(* CoDeSys 2.3 library: Mio_plc.lib *)

(* Global variable list: Globale_Variablen *)
(*
 PLC1131-Library with Functions to M-IO-Handler and IO-Hardware
 Copyright: G.Bachmann GmbH, 1997-2017, Feldkirch - Austria
*)
VAR_GLOBAL CONSTANT
	MIO_PLC_LIBVER					:	STRING(16) 	:=	'V1.39 Release';	(* Version String *)
    MIO_PLC_MMPREADY                :   BOOL        :=  TRUE;               (* MMP Ready *)

	(* Error-Return-Codes *)
	(* ATTENTION: actual Codes must be interpreted (modulo 1000)! *)
	Mio_ERC_Other:			DINT := -1;			(* MIO-Function unsuccessfull *)
	Mio_ERC_ParmInvalid:	DINT := -2;			(* Parameters are invalid *)
	Mio_ERC_NoCard:			DINT := -3;			(* Card not found / existing *)
	Mio_ERC_NoSelf:			DINT := -8;			(* Caller is no PLC *)
	Mio_ERC_Other2:			DINT := -9;			(* MIO-Function unsuccessfull *)
    Mio_ERC_NoMemory:       DINT := -10;		(* Memory can't be allocated *)
	Mio_ERC_Internal:		DINT := -11;		(* Internal Error *)

	(* Constants used with Mio...Select *)
	Mio_OBJ_AllChan:		DWORD := 16#80000000;
	Mio_OBJ_Card:			DWORD := 16#80000001;

    (* possible values for Card-Mode *)
    MIO_MODE_REAL:          DINT := 1;          (* IO-Module is present *)
    MIO_MODE_VIRTUAL:       DINT := 2;          (* IO-Module is virtuel *)
    MIO_MODE_VIRTSIM:       DINT := 3;          (* @deprecated IO-Module has simulated values *)
    MIO_MODE_REALFB:        DINT := 4;          (* IO-Module AT fieldbus *)
    MIO_MODE_VIRTUALRW:     DINT := 5;          (* virtual IO-Module, writeable inputs *)
    MIO_MODE_REALSRV:       DINT := 6;          (* IO-Module connected TO a service *)
    MIO_MODE_VIRTUALSRV:    DINT := 7;          (* IO-Module connected TO a service *)

	(* Constants used as Card-Type *)
	Mio_TYP_MP213:			DINT := 1; 		(* Module of type MP213 *)
	Mio_TYP_MP2XX:			DINT := 1; 		(* Module of type MP2XX *)
	Mio_TYP_DI216:			DINT := 2; 		(* Module of type DI216 *)
	Mio_TYP_DO216:			DINT := 3; 		(* Module of type DO216 *)
	Mio_TYP_DI232:			DINT := 4; 		(* Module of type DI232 *)
	Mio_TYP_DO232:			DINT := 5; 		(* Module of type DO232 *)
	Mio_TYP_AI204:			DINT := 6; 		(* Module of type AI204 *)
	Mio_TYP_AO202:			DINT := 7; 		(* Module of type AO202 *)
	Mio_TYP_ISI202:			DINT := 8; 		(* Module of type ISI202 *)
	Mio_TYP_AIO288:			DINT := 9; 		(* Module of type AIO288 *)
	Mio_TYP_FBM201:			DINT := 10; 	(* Module of type FM201 *)
	Mio_TYP_FBS202:			DINT := 11;		(* Module of type FS202 *)
	Mio_TYP_CM202:			DINT := 12;		(* Module of type CM202 *)
	Mio_TYP_BEM201:			DINT := 13;		(* Module of type BEM201 *)
	Mio_TYP_BES202:			DINT := 14;		(* Module of type BES202 *)
	Mio_TYP_ACR222:			DINT := 15;		(* Module of type ACR222 *)
	Mio_TYP_ME203:			DINT := 16;		(* Module of type ME203 *)
	Mio_TYP_CS200:			DINT := 17;		(* Module of type CS200 *)
	Mio_TYP_RS204:			DINT := 18;		(* Module of type RS204 *)
	Mio_TYP_DMS202:			DINT := 19;		(* Module of type DMS202 *)
	Mio_TYP_NT230:			DINT := 20;		(* Module of type NT230 *)
	Mio_TYP_DIO216:			DINT := 21;		(* Module of type DIO216 *)
	Mio_TYP_DI212:			DINT := 24;		(* Module of type DI212 *)
	Mio_TYP_DIO264_C:		DINT := 25;		(* Module of type DIO16/32/48/64_C *)
	Mio_TYP_BS2XX:			DINT := 26;		(* Bus Module of type BS2XX *)
	Mio_TYP_FM21X:			DINT := 27;		(* Module of type FM211, FM212 *)
	Mio_TYP_FS21X:			DINT := 28;		(* Module of type FS211, FS212 *)
	Mio_Typ_FM2XX:   		DINT := 27; 	(* Module of type FM211, FM212, FM221, FM222 *)
	Mio_Typ_FS2XX:   		DINT := 28;  	(* Module of type FS211, FS212, FS221, FS222 *)
	Mio_TYP_ES200:			DINT := 29;		(* Module of type ES200 *)
	Mio_TYP_DPM200:			DINT := 30;		(* Module of type DPM200 *)
	Mio_TYP_CNT204:			DINT := 31;		(* Module of type CNT204 *)
	Mio_TYP_PTAI216:		DINT := 32;		(* Module of type PTAI216 *)
	Mio_TYP_PWM202:			DINT := 33;		(* Module of type PWM202 *)
	Mio_TYP_TCO216_C:		DINT := 34;		(* Module of type TCO216-C *)
	Mio_TYP_AO208:			DINT := 35;		(* Module of type AO208 *)
	Mio_TYP_DIO280:			DINT := 36;		(* Module of type DIO248/64/80 *)
	Mio_TYP_DIO2XX:			DINT := 36;		(* Module of type DIO248/64/80 *)
	Mio_TYP_TTL264:			DINT := 37;		(* Module of type TTL264 *)
	Mio_TYP_SEM201:         DINT := 38;     (* Module of type SEM201 *)
	Mio_TYP_IOP201:         DINT := 39;     (* Module of type IOP201 *)
    Mio_TYP_BSI200:         DINT := 40;     (* Module of type BSI200 (no drv) *)
    Mio_TYP_MTS200:         DINT := 41;     (* Module of type MTS200 (no drv) *)
    Mio_TYP_PCFS212:        DINT := 42;     (* Module of type PCFS212 *)
    Mio_TYP_DNM201:         DINT := 43;     (* Module of type DNM201 *)
	Mio_TYP_AI20XSI:		DINT := 44;		(* Module of type AI20X/SI *)
	Mio_TYP_AO20XSI:		DINT := 45;		(* Module of type AO20X/SI *)
    Mio_TYP_WT305E:         DINT := 46;     (* Module of type WT305e (no drv) *)
	Mio_TYP_EM203:			DINT := 47; 	(* Module of type EM203 *)
	Mio_TYP_MPC2XX:			DINT := 49; 	(* Module of type MPC2XX *)
	Mio_TYP_MX2XX:			DINT := 50;		(* Module of type MX2XX *)
	Mio_TYP_WT3XX:          DINT := 51;     (* Module of type WT3XX (no drv) *)
    Mio_TYP_PCM201:         DINT := 52;     (* Internal Module (no drv) *)
    Mio_TYP_DIO232:         DINT := 53;     (* Module of type DIO232 *)
    Mio_TYP_BET200:         DINT := 54;     (* Internal Module (no drv) *)
    Mio_TYP_PN201:          DINT := 55;     (* Module of type PN201 *)
    Mio_TYP_NT255:          DINT := 56;     (* Module of type NT255 *)
    Mio_TYP_MBM201:         DINT := 57;     (* Module of type Modbus Master *)
    Mio_TYP_WT2XX:          DINT := 58;     (* Module of type WT2XX (no drv) *)
    Mio_TYP_CT2XX:          DINT := 59;     (* Module of type CT2XX *)
    Mio_TYP_DA3284C:        DINT := 60;     (* Module of type DA3284C *)
	Mio_TYP_AIC2XX:         DINT := 61;     (* Module of type AIC2XX *)
	Mio_TYP_CAN:            DINT := 62;     (* Logical CAN Module *)
	Mio_TYP_ECAT201:        DINT := 63;     (* Module of type ECAT201 *)
	Mio_TYP_TI214:          DINT := 64;     (* Module of type TI214 *)
	Mio_TYP_EVALBOARD:      DINT := 65;     (* HW Evaluation Board *)
	Mio_TYP_PN23:           DINT := 66;     (* PCI Module of type PN23 ProfiNet IRT *)
    Mio_TYP_OT100:          DINT := 67;     (* OT100 Terminal *)
    Mio_TYP_SLC284:         DINT := 68;     (* Module OF TYPE SLC284 *)
    Mio_TYP_SDI208:         DINT := 69;     (* Module OF TYPE SDI208 *)
    Mio_TYP_SDO204:         DINT := 70;     (* Module OF TYPE SDO204 *)
	Mio_TYP_ETH2X:          DINT := 77;     (* Module of type ETH2X *)
	Mio_TYP_DOR206:         DINT := 78;     (* Module of type DOR206 *)
	Mio_TYP_DMW200:         DINT := 79;     (* Module of Drive-Middleware *)
	Mio_TYP_SERCOS:         DINT := 80;     (* Module of Drive-Middleware *)
	Mio_TYP_AP211:          DINT := 81;     (* Module of type AP21X *)
	Mio_TYP_MH2XX:          DINT := 82;     (* Module of type MH2XX *)
	Mio_TYP_MMSCNLT:        DINT := 83;     (* Module of type MMS-Client *)
	Mio_TYP_SFS240C:        DINT := 84;     (* Module of type SFS240C *)
	Mio_TYP_FCS2XX:         DINT := 85;     (* Module of type FCS2xx *)
	Mio_TYP_CT1300:         DINT := 86;     (* Module of type CT1300 *)
	Mio_TYP_OT1300:         DINT := 87;     (* Module of type OT1300 *)
	Mio_TYP_AI208SI:        DINT := 88;     (* Module of type AI208/SI *)
	Mio_TYP_GMP232:         DINT := 89;     (* Module of type GMP232 *)
    Mio_TYP_BCP200:         DINT := 90;     (* Module OF TYPE BCP200 *)
    Mio_TYP_BCH200:         DINT := 91;     (* Module OF TYPE BCH200 *)
    Mio_TYP_EM213:          DINT := 92;     (* Module OF TYPE EM213 *)
    Mio_TYP_ECS200:         DINT := 93;     (* Module OF TYPE ECS200 *)
    Mio_TYP_BCP202:         DINT := 94;     (* Module OF TYPE BCP202 *)
    Mio_TYP_BCH202:         DINT := 95;     (* Module OF TYPE BCH202 *)
    Mio_TYP_BCR202:         DINT := 96;     (* Module OF TYPE BCR202 *)
    Mio_TYP_MC2XX:          DINT := 97;     (* Module OF TYPE MC2XX *)
    Mio_TYP_MBUS:           DINT := 98;     (* Service OF TYPE MBUS *)
	MIO_TYP_GIO2XX:         DINT := 99;     (* Service OF TYPE GIO2XX *)
	MIO_TYP_GSP274:         DINT := 100;    (* Module OF TYPE GSP274 *)
	MIO_TYP_S60870_5:       DINT := 101;    (* Module OF TYPE IEC 60870-5-104 server *)
    MIO_TYP_AIO2XX:         DINT := 102;    (* Module of type AIO2XX *)
	MIO_TYP_SVMXXX:     	DINT := 103;    (* Module of type SVMXXX *)
	MIO_TYP_OPCUAS:      	DINT := 104;    (* Module of type OPCUAS *)
	MIO_TYP_BPC600:       	DINT := 105;    (* Module of type BCP600 *)
	MIO_TYP_STMI3XX:      	DINT := 106;    (* Module of type STMI3XX *)
	MIO_TYP_GM260:       	DINT := 107;    (* Module of type GM260 *)
	MIO_TYP_CPC2XX:         DINT := 108;    (* CompactPLC of type CPC2xx *)
	MIO_TYP_CAIO284:        DINT := 109;    (* AIO284 for CPC2XX *)
	MIO_TYP_CISI2XX:     	DINT := 110;    (* ISI2XX for CPC2XX *)
	MIO_TYP_CDIO2XX:        DINT := 111;    (* DIO2XX for CPC2XX *)
	MIO_TYP_GM2XX:      	DINT := 112;    (* Module of type GM2XX (GM210 and GM230) *)
	MIO_TYP_OT1200:       	DINT := 113;    (* Module of type OT1200 *)
	MIO_TYP_MR2XX:        	DINT := 114;  	(* Module of type MR2XX *)
	MIO_TYP_DIOXXC:       	DINT := 115;    (* Module of type DIOxx-C Standalone CAN-Modules *)
	MIO_TYP_AIO2XXSI:     	DINT := 116;    (* Module of type AIO2XX/SI *)
	MIO_TYP_DNP3:         	DINT := 117;   	(* Service of type DNP3 *)
	MIO_TYP_SCT202:         DINT := 118;    (* Module of type SCT202 *)
	MIO_TYP_GMP232X:      	DINT  := 119;   (* Module of type GMP232/X *)
	MIO_TYP_PVA2XX:       	DINT  := 120;   (* Module of type PVA2XX *)
	MIO_TYP_TSTDRV:       	DINT  := 254;   (* Generic ID for test drivers *)

    (* Constants used as Card-Variant *)

	(* in case of type MIO_TYP_MP2XX *)
	MIO_V_MP213:    DINT  := 0;     (* Module of type MP213 *)
	MIO_V_MP226:    DINT  := 1;     (* Module of type MP226 *)
	MIO_V_MP236:    DINT  := 2;     (* Module of type MP236 *)
	MIO_V_MP240:    DINT  := 3;     (* Module of type MP240 *)
	MIO_V_MP213EW:  DWORD := 16#20; (* Module of type MP213/EW *)
	MIO_V_MP226EW:  DWORD := 16#21; (* Module of type MP226/EW *)

	(* in case of type MIO_TYP_ME203 *)
	MIO_V_ME203:    DINT  := 0;     (* Module of type ME203 *)
	MIO_V_ME203N:   DINT  := 1;     (* Module of type ME203/N *)
	MIO_V_ME203C:   DINT  := 2;     (* Module of type ME203/C *)
	MIO_V_ME203CN:  DINT  := 3;     (* Module of type ME203/CN *)
	MIO_V_ME203E:   DINT  := 4;     (* Module of type ME203/E *)
	MIO_V_ME203EN:  DINT  := 5;     (* Module of type ME203/EN *)
	MIO_V_ME203CNW: DWORD := 16#23; (* Module of type ME203/CNW *)

	(* WT/CT Version in case of type Mio_TYP_WTXXX for 200 and 300 series. *)
	MIO_VF_DISPLAYMASK: DWORD := 16#0f;         (* filter for display type *)
	MIO_VF_DIMMABLE:    DWORD := 16#10;         (* dimmable display *)
	MIO_VF_IRTOUCH:     DWORD := 16#40;         (* IR Touch *)
	MIO_VF_ALARM:       DWORD := 16#80;         (* has extern alarm IOs *)
	MIO_V_WT305:        DINT  := 0;             (* Module of type WT305 1/4 VGA *)
	MIO_V_WT306:        DINT  := 1;             (* Module of type WT306 VGA *)
	MIO_V_WT310:        DINT  := 2;             (* Module of type WT310 *)
	MIO_V_WT312:        DINT  := 3;             (* Module of type WT312 *)
	MIO_V_WT315:        DINT  := 4;             (* Module of type WT315 *)
	MIO_V_WT317:        DINT  := 5;             (* Module of type WT317 *)
	MIO_V_WT319:        DINT  := 6;             (* Module of type WT319 *)
	MIO_V_WT305V:       DINT  := 7;             (* Module of type WT305V *)
	MIO_V_CT305:        DINT  := MIO_V_WT305;   (* Module of type CT305 1/4 VGA *)
	MIO_V_CT306:        DINT  := MIO_V_WT306;   (* Module of type CT306 VGA *)
	MIO_V_CT310:        DINT  := MIO_V_WT310;   (* Module of type CT310 *)
	MIO_V_CT312:        DINT  := MIO_V_WT312;   (* Module of type CT312 *)
	MIO_V_CT315:        DINT  := MIO_V_WT315;   (* Module of type CT315 *)
	MIO_V_CT317:        DINT  := MIO_V_WT317;   (* Module of type CT317 *)
	MIO_V_CT319:        DINT  := MIO_V_WT319;   (* Module of type CT319 *)
	MIO_V_CT305V:       DINT  := MIO_V_WT305V;  (* Module of type CT305 VGA *)
	MIO_V_WT205:        DINT  := MIO_V_WT305;   (* Module of type WT205 1/4 VGA *)
	MIO_V_WT205V:       DINT  := MIO_V_WT305V;  (* Module of type WT205 VGA *)
	MIO_V_CT205:        DINT  := MIO_V_WT205;   (* Module of type CT205 1/4 VGA *)
	MIO_V_CT205V:       DINT  := MIO_V_WT205V;  (* Module of type CT205 VGA *)
	MIO_V_CT205M:       DWORD := 16#00000097;

	(* in case of type MIO_TYP_MPC2XX *)
	MIO_V_MPC240:   DINT  := 0;     (* Module of type MPC240 *)
	MIO_V_MPC265:   DINT  := 1;     (* Module of type MPC265 *)
	MIO_V_MPC270:   DINT  := 2;     (* Module of type MPC270 *)
	MIO_V_MPC293:   DINT  := 3;     (* Module of type MPC293 *)
	MIO_V_MPC240CW: DWORD := 16#20; (* Module of type MPC240/CW *)
	MIO_V_MPC265CW: DWORD := 16#21; (* Module of type MPC265/CW *)
	MIO_V_MPC270CW: DWORD := 16#22; (* Module of type MPC270/CW *)
	MIO_V_MPC293CW: DWORD := 16#23; (* Module of type MPC293/CW *)

	(* in case of type MIO_TYP_MPC2XX (MPE2xx CPUs) *)

	MIO_V_MPE2XX:   DWORD := 16#10; (* Module of type MPE2xx *)
	MIO_V_MPE240:   DWORD := 16#10; (* Module of type MPE240 *)
	MIO_V_MPE265:   DWORD := 16#11; (* Module of type MPE265 *)
	MIO_V_MPE270:   DWORD := 16#12; (* Module of type MPE270 *)

	(* in case of type MIO_TYP_MX2XX *)
	MIO_VF_MX2xx_N:     DWORD := 16#01;         (* MX2xx bitmask: has integrated power supply *)
	MIO_VF_MX2xx_CW:    DWORD := 16#20;         (* MX2xx bitmask: is a cold weather variant *)
	MIO_V_MX213:        DWORD := 16#00;         (* MX2xx bitmask: Module of type MX213 *)
	MIO_V_MX213N:       DWORD := 16#00000001;
	MIO_V_MX213CW:      DWORD := 16#00000020;
	MIO_V_MX213NCW:     DWORD := 16#00000021;
	MIO_V_MX207:        DWORD := 16#02;         (* MX2xx bitmask: Module of type MX207 *)
	MIO_V_MX207N:       DWORD := 16#00000003;
	MIO_V_MX207CW:      DWORD := 16#00000022;
	MIO_V_MX207NCW:     DWORD := 16#00000023;
	MIO_V_MX220:        DWORD := 16#04;         (* MX2xx bitmask: Module of type MX220 *)
	MIO_V_MX220N:       DWORD := 16#00000005;
	MIO_V_MX220CW:      DWORD := 16#00000024;
	MIO_V_MX220NCW:     DWORD := 16#00000025;

	(* in case of type MIO_TYP_MH2XX *)
	MIO_V_MH212S:   DINT  := 0; (* Module of type MH212/S *)
	MIO_V_MH212:    DINT  := 1; (* Module of type MH212 *)
	MIO_V_MH230:    DINT  := 2; (* Module of type MH230 *)

	(* in case of type MIO_TYP_MC2XX *)
	MIO_V_MC205:    DINT  := 0; (* Module of type MC205 (600MHz) *)
	MIO_V_MC210:    DINT  := 1; (* Module of type MC210 (1600MHz) *)
	MIO_V_MC206:    DINT  := 2; (* Module OF TYPE MC206 (Single core 800MHz) *)
	MIO_V_MC212:    DINT  := 3; (* Module OF TYPE MC212 (Dual core 1300MHz) *)
	MIO_V_MC220:    DINT  := 4; (* Module OF TYPE MC220 (Quad core 1600MHz) *)

	(* in case of type MIO_TYP_ISI2xx *)
	MIO_V_ISI222:   DWORD := 16#81; (* Module of type ISI222 *)

	(* in case of type MIO_TYP_DIOXXC *)
	MIO_V_DIO43C:   DWORD := 16#00; (* Module of type DIO43-C *)
	MIO_V_DIO62C:   DWORD := 16#01; (* Module of type DIO62-C *)

	(* in case of type MIO_TYP_CPC2XX *)
	MIO_V_CPC210:   DWORD := 16#01; (* Module of type CPC210 *)

	(* in case of type MIO_TYP_MR2XX *)
	MIO_V_MR201:    DWORD := 16#00; (* Module of type MR201 *)
	MIO_V_MR202:    DWORD := 16#01; (* Module of type MR202 *)

	(* in case of type MIO_TYP_GM2XX *)
	MIO_V_GM230:    DWORD := 16#00; (* Module of type GM230 *)
	MIO_V_GM210:    DWORD := 16#01; (* Module of type GM210 *)

	(* in case of type MIO_TYP_GMP232X *)
	MIO_V_GMP232_1: DWORD := 16#01; (* Module of type GMP232/1 *)
	MIO_V_GMP232_2: DWORD := 16#02; (* Module of type GMP232/2 *)
	MIO_V_GMP232_3: DWORD := 16#03; (* Module of type GMP232/3 *)
	MIO_V_GMP232_4: DWORD := 16#04; (* Module of type GMP232/4 *)

    (* Constants used as Card- and Channel-Category *)
	Mio_CTG_Di:				DWORD := 16#0001; 		(* Card/Chan with DI capability *)
	Mio_CTG_Do:				DWORD := 16#0002; 		(* Card/Chan with DO capability *)
	Mio_CTG_Ai:				DWORD := 16#0004; 		(* Card/Chan with AI capability *)
	Mio_CTG_Ao:				DWORD := 16#0008; 		(* Card/Chan with AO capability *)
	Mio_CTG_Inc:			DWORD := 16#0010; 		(* Card/Chan with INC capability *)
	Mio_CTG_Ssi:			DWORD := 16#0020; 		(* Card/Chan with SSI capability *)
	Mio_CTG_Drive:			DWORD := 16#0040; 		(* Card/Chan for drives *)
	Mio_CTG_Interface:		DWORD := 16#0080; 		(* Card/Chan with an interface *)
	Mio_CTG_Count:			DWORD := 16#0100; 		(* Card/Chan with CNT capability *)
	Mio_CTG_Trigg:			DWORD := 16#0200; 		(* Card/Chan with TRG capability *)
	Mio_CTG_Pwm:			DWORD := 16#0400; 		(* Card/Chan with PWM capability *)
	Mio_CTG_Freq:			DWORD := 16#0800; 		(* Card/Chan with FREQ capability *)
	Mio_CTG_Stat:			DWORD := 16#1000; 		(* Card/Chan with Status cap. *)
	Mio_CTG_Cntrl:			DWORD := 16#2000; 		(* Card/Chan with Control cap. *)
	Mio_CTG_Time:			DWORD := 16#8000;		(* Card/Chan with time measure cap. *)
	Mio_CTG_Diff: 			DWORD := 16#10000;		(* Card/Chan with diff. measure cap. *)
    Mio_CTG_Velocity:       DWORD := 16#20000;      (* Card with velocity measure cap. *)
	Mio_CTG_Bes:			DWORD := 16#04000000; 	(* Card is Bus Extension Slave *)
	Mio_CTG_Bem:			DWORD := 16#08000000; 	(* Card is Bus Extension Master *)
	Mio_CTG_Cpu:			DWORD := 16#10000000; 	(* CPU module *)
	Mio_CTG_Fbs:			DWORD := 16#20000000; 	(* Card with FastBusSlave cap. *)
	Mio_CTG_Fbm:			DWORD := 16#40000000; 	(* Card with FastBusMaster cap. *)
	Mio_CTG_FB:				DWORD := 16#80000000; 	(* Card with Fieldbus capability *)

	(* Constants used as Card- and Channel-Flags *)
	Mio_FLG_Read:			DWORD := 16#0001; 		(* Card/Chan is readable *)
	Mio_FLG_Write:			DWORD := 16#0002; 		(* Card/Chan is writable *)
	Mio_FLG_RW:				DWORD := 16#0003; 		(* Card/Chan is read-/writable *)
	Mio_FLG_Error:			DWORD := 16#0004; 		(* Card/Chan has error interrupt *)
	Mio_FLG_Event:			DWORD := 16#0008; 		(* Card/Chan has event interrupt *)
	Mio_FLG_Select:			DWORD := 16#0010; 		(* Card/Chan has select functions *)
	Mio_FLG_BadIO: 			DWORD := 16#0400; 		(* Card has been deactivated *)
	Mio_FLG_Fnled:			DWORD := 16#0800; 		(* Card has function for LED flashing *)
	Mio_FLG_Bcheck:			DWORD := 16#1000; 		(* Card supports IO-Bus check *)
	Mio_FLG_Acheck:			DWORD := 16#2000; 		(* Card supports Alive check *)
	Mio_FLG_Watchdog:		DWORD := 16#4000; 		(* Card has watchdog to be triggered *)
	Mio_FLG_Firmware:		DWORD := 16#8000; 		(* Card has firmware or updatable logic on it *)
	Mio_FLG_SVar:			DWORD := 16#200000;		(* Card has service variables *)
	Mio_FLG_HwPiReady:		DWORD := 16#400000;		(* Card is ready for hardware process image *)
	Mio_FLG_HwPiSupp:		DWORD := 16#800000;		(* Card supports hardware process image *)
	Mio_FLG_FIFOVar:		DWORD := 16#1000000;	(* Card supports variable FIFO flush address *)
	Mio_FLG_ChPiSupp:		DWORD := 16#2000000;	(* Card supports selected channel process image *)

	(* Constants used for Error-State *)
	Mio_ERR_Badstation:		DWORD := 16#0001; 		(* Module is on Bad Station *)
	Mio_ERR_Power:			DWORD := 16#0002;		(* Ext./int. power failure *)
	Mio_ERR_BrokenWire:		DWORD := 16#0004;		(* Open In/Out circuit *)
	Mio_ERR_ShortCirc:		DWORD := 16#0008;		(* Short In/Out circuit *)
	Mio_ERR_TempTooHi:		DWORD := 16#0010;		(* Temperatue too high *)
	Mio_ERR_Decoder:		DWORD := 16#0020;		(* Decoder/Encoder error *)
	Mio_ERR_Accu:			DWORD := 16#0040;		(* @deprecated Battery voltage low *)
    Mio_ERR_ChanDisabled:   DWORD := 16#0040;       (* Channel is disabled *)
	Mio_ERR_Init:			DWORD := 16#0080;		(* @deprecated Error in init function *)
	Mio_ERR_BadConfig:		DWORD := 16#0080;		(* Configuration not valid *)
	Mio_ERR_Watchdog:		DWORD := 16#0100;		(* Internal watchdog error *)
	Mio_ERR_External:		DWORD := 16#0200;		(* External error *)
	Mio_ERR_Ready:			DWORD := 16#0400;		(* @deprecated Modul internal cycle done *)
	Mio_ERR_Dead: 			DWORD := 16#0400; 		(* Module alive test failed *)
	Mio_ERR_OutDisabled:	DWORD := 16#0800;		(* Output is disabled *)
	Mio_ERR_Voltagetohi:	DWORD := 16#1000;		(* External voltage too high *)
	Mio_ERR_Voltagetolo:	DWORD := 16#2000;		(* External voltage too low *)
	Mio_ERR_Currenttohi:	DWORD := 16#4000;		(* Output current too high *)
	Mio_ERR_Badprofile:		DWORD := 16#00008000; 	(* Profile not valid *)
	Mio_ERR_MaskSystem:		DWORD := 16#0000FFFF;	(* Generic errors *)
	Mio_ERR_MaskUser:		DWORD := 16#FFFF0000;	(* Driver specific error *)

	(* Constants used for Event-State *)
	Mio_EVT_Value:			DWORD := 16#0001;		(* Event on change OF value *)
	Mio_EVT_Reference:		DWORD := 16#0002;		(* Event AT reference point *)
	Mio_EVT_Reset:			DWORD := 16#0004;		(* Event home done *)
	Mio_EVT_Latchstrb:		DWORD := 16#0010;		(* Latch into strobe register done *)
	Mio_EVT_Latchref:		DWORD := 16#0020;		(* Latch into reference register done *)
	Mio_EVT_Latchstrbov:	DWORD := 16#0040;		(* Latch strobe overwritten *)
	Mio_EVT_Latchreflos:	DWORD := 16#0080;		(* Latch referenz register lost *)

	(* Constants used as Error-State in case of SSI-Inputs *)
	Mio_ERR_Clock:			DWORD := 16#00010000;

   (* Possible driver specific error for PWM module *)
	MIO_ERR_MAXCURRENT:   DWORD := 16#00040000;   (* Max. current reached *)

   (* Possible driver specific error for PCFS module *)
	MIO_ERR_TRANSMIT: DWORD := 16#00100000;   (* Data transmission error *)
	MIO_ERR_PCIRESET: DWORD := 16#00200000;   (* PCI-Reset *)

   (* Possible driver specific error for AI204/SI module *)
	MIO_ERR_POSRANGE:     DWORD := 16#00400000;   (* Value above maximum *)
	MIO_ERR_NEGRANGE:     DWORD := 16#00800000;   (* Value below minimum *)
	MIO_ERR_MONITORING:   DWORD := 16#01000000;   (* Monitoring error! *)

    (* Possible driver specific error for Safety modules *)
    Mio_ERR_SafetyGenErr:   DWORD := 16#00010000;    (* General module error *)

	(* Possible driver specific errors for MBM201 modules *)
	MIO_ERR_CONNECTION:       DWORD := 16#00000400;   (* No connection *)
	MIO_ERR_EXCEPTION:        DWORD := 16#00010000;   (* Modbus exception *)
	MIO_ERR_CYCLETIMETOOLONG: DWORD := 16#00020000;   (* Cycle time too long *)
	MIO_ERR_CRCERROR:         DWORD := 16#00040000;   (* CRC error *)

   (* Possible driver specific errors/warning for FM2XX/FS2XX, FCS2XX modules *)
	MIO_WRN_LINE_A:     DWORD := 16#00010000;   (* FO Line A RX Power has critical level. *)
	MIO_ERR_LINE_A:     DWORD := 16#00020000;   (* FO Line A RX Power is below critical level. *)
	MIO_WRN_LINE_B:     DWORD := 16#00100000;   (* FO Line B RX Power has critical level. *)
	MIO_ERR_LINE_B:     DWORD := 16#00200000;   (* FO Line B RX Power is below critical level. *)
	MIO_ERR_TRIGGER_A:  DWORD := 16#01000000;   (* FO Line A user defined triggervalue *)

    (* ECS200 specific error and event interrupts *)
    MIO_ERR_ECSGENERR:      DWORD := 16#00010000;     (* General module error *)
    MIO_EVT_ECSSYNC0:       DWORD := 16#00010000;     (* SYNC0 Event *)
    MIO_EVT_ECSSYNC1:       DWORD := 16#00020000;     (* SYNC1 Event *)

    (* DIO2xx specific error and event interrupts *)
    MIO_ERR_PWFMODULE:      DWORD := 16#00020000;     (* Power fail complete module *)
    MIO_ERR_PHASE:          DWORD := 16#00040000;     (* Phase error *)
    MIO_EVT_OVERFLOW:       DWORD := 16#02000000;     (* Value overflow *)

    (* GIO212, AIO216 and AIO208 specific error and event interrupts *)
	MIO_ERR_LOWERRANGE:   DWORD := 16#00010000;       (* Lowerrange exceeded *)
	MIO_ERR_UPPERRANGE:   DWORD := 16#00020000;       (* Upperrange exceeded *)
	MIO_EVT_REFERENCE2:   DWORD := 16#00010000;       (* Second reverence value reached *)
    MIO_EVT_LOWERLIMIT:   DWORD := 16#00020000;       (* Lower LIMIT reached *)
    MIO_EVT_UPPERLIMIT:   DWORD := 16#00040000;       (* Upper LIMIT reached *)

   (* Events for SCT202 module *)
    MIO_EVT_OVERSPEED:    DWORD := 16#00010000;       (* Chan 1-4 *)
    MIO_EVT_STAGNATION:   DWORD := 16#00020000;       (* Chan 1-4 *)

	(* RS204 specific event interrupts *)
	MIO_EVT_POWER_UART1:  DWORD := 16#00010000;   	(* Powerfail UART1 *)
	MIO_EVT_POWER_UART2:  DWORD := 16#00020000;   	(* Powerfail UART2 *)
	MIO_EVT_POWER_UART3:  DWORD := 16#00040000;   	(* Powerfail UART3 *)
	MIO_EVT_POWER_UART4:  DWORD := 16#00080000;   	(* Powerfail UART4 *)

	(* GMP232X specific event flags. None of them are shared with the standard GMP232. *)
	MIO_EVT_QU_PCC1:     DWORD := 16#00000002;   (* QU PCC1 *)
	MIO_EVT_QU_PCC2:     DWORD := 16#00000004;   (* QU PCC2 *)
	MIO_EVT_ANYZERO:     DWORD := 16#00000010;   (* Any voltage zero crossing *)
	MIO_EVT_P1ZERO:      DWORD := 16#00000020;   (* Phase 1 voltage positive zero crossing *)
	MIO_EVT_SCOPE:       DWORD := 16#00000040;   (* Scope event *)
	MIO_EVT_HEARTBEAT:   DWORD := 16#00000080;   (* Heartbeat (module health check) *)
	MIO_EVT_REV_POWER1:  DWORD := 16#00000100;   (* Rev. power 1 *)
	MIO_EVT_REV_POWER2:  DWORD := 16#00000200;   (* Rev. power 2 *)
	MIO_EVT_HARM_U:      DWORD := 16#00008000;   (* Voltage harmonics *)
	MIO_EVT_U_ASYM1:     DWORD := 16#00010000;   (* Voltage asymmetry 1 *)
	MIO_EVT_U_ASYM2:     DWORD := 16#00020000;   (* Voltage asymmetry 2 *)
	MIO_EVT_THD_U:       DWORD := 16#00040000;   (* Voltage THD *)
	MIO_EVT_I_ASYM1:     DWORD := 16#00080000;   (* Current asymmetry 1 *)
	MIO_EVT_I_ASYM2:     DWORD := 16#00100000;   (* Current asymmetry 2 *)
	MIO_EVT_HARM_I:      DWORD := 16#00200000;   (* Current harmonics *)
	MIO_EVT_VECTORJUMP1: DWORD := 16#00400000;   (* Vector jump 1 *)
	MIO_EVT_VECTORJUMP2: DWORD := 16#00800000;   (* Vector jump 2 *)
	MIO_EVT_TDD_I:       DWORD := 16#01000000;   (* TDD *)
	MIO_EVT_DIRCURRENT1: DWORD := 16#02000000;   (* Directional overcurrent 1 *)
	MIO_EVT_DIRCURRENT2: DWORD := 16#04000000;   (* Directional overcurrent 2 *)
	MIO_EVT_ROCOF:       DWORD := 16#08000000;   (* ROCOF *)
	MIO_EVT_MAX_POWER1:  DWORD := 16#10000000;   (* Maximal power 1 *)
	MIO_EVT_MAX_POWER2:  DWORD := 16#20000000;   (* Maximal power 2 *)
	MIO_EVT_MANUAL_REL1: DWORD := 16#40000000;   (* State of manual relay 1 *)
	MIO_EVT_MANUAL_REL2: DWORD := 16#80000000;   (* State of manual relay 2 *)

	(* GMP232X specific error interrupts *)
	MIO_ERR_NEGSYS_HI:      DWORD := 16#00000008;   (* Negative system blocking upper limit *)
	MIO_ERR_V_LO1:          DWORD := 16#00000010;   (* Voltage lower limit 1 *)
	MIO_ERR_V_LO2:          DWORD := 16#00000020;   (* Voltage lower limit 2 *)
	MIO_ERR_V_HI4:          DWORD := 16#00000100;   (* Voltage upper limit 4 (supported for FW >= 1.03R) *)
	MIO_ERR_V_LO3:          DWORD := 16#00000200;   (* Voltage lower limit 3 *)
	MIO_ERR_V_LO4:          DWORD := 16#00000800;   (* Voltage lower limit 4 (supported for FW >= 1.03R) *)
	MIO_ERR_V_HI1:          DWORD := 16#00001000;   (* Voltage upper limit 1 *)
	MIO_ERR_V_HI2:          DWORD := 16#00002000;   (* Voltage upper limit 2 *)
	MIO_ERR_V_HI3:          DWORD := 16#00004000;   (* Voltage upper limit 3 *)
	MIO_ERR_VFRT1:          DWORD := 16#00008000;   (* Voltage FRT 1 *)
	MIO_ERR_VFRT2:          DWORD := 16#00010000;   (* Voltage FRT 2 *)
	MIO_ERR_VFRT3:          DWORD := 16#00020000;   (* Voltage FRT 3 *)
	MIO_ERR_VFRT4:          DWORD := 16#00040000;   (* Voltage FRT 4 *)
	MIO_ERR_I_HI1:          DWORD := 16#00080000;   (* Current upper limit 1 *)
	MIO_ERR_I_HI2:          DWORD := 16#00100000;   (* Current upper limit 2 *)
	MIO_ERR_I_HI3:          DWORD := 16#00200000;   (* Current upper limit 3 *)
	MIO_ERR_QU_GEN1:        DWORD := 16#00400000;   (* QU limit 1 *)
	MIO_ERR_QU_GEN2:        DWORD := 16#00800000;   (* QU limit 2 *)
	MIO_ERR_FFRT1:          DWORD := 16#01000000;   (* Frequency FRT 1 *)
	MIO_ERR_FFRT2:          DWORD := 16#02000000;   (* Frequency FRT 2 *)
	MIO_ERR_F_HI3:          DWORD := 16#04000000;   (* Frequency upper limit 3 *)
	MIO_ERR_F_HI2:          DWORD := 16#08000000;   (* Frequency upper limit 2 *)
	MIO_ERR_F_HI1:          DWORD := 16#10000000;   (* Frequency upper limit 1 *)
	MIO_ERR_F_LO3:          DWORD := 16#20000000;   (* Frequency lower limit 3 *)
	MIO_ERR_F_LO2:          DWORD := 16#40000000;   (* Frequency lower limit 2 *)
	MIO_ERR_F_LO1:          DWORD := 16#80000000;   (* Frequency lower limit 1 *)
	MIO_ERR_MSK_GMP232X:    DWORD := 16#FFFFFB38;   (* For all other error bits see generic MIO errors (Flags for 1.03R included) *)

	(* Constants used as Channel-Mode for DIO2xx  *)
	Mio_MODE_In:			DWORD := 16#0001;		(* Channel is input *)
	Mio_MODE_Out:			DWORD := 16#0002;		(* Channel is output *)
	Mio_MODE_InOutMsk:		DWORD := 16#0003; 		(* Mask for IN and OUT *)
	Mio_MODE_PosEdge:		DWORD := 16#0010;
	Mio_MODE_NegEdge:		DWORD := 16#0020;
	Mio_MODE_BothEdges:		DWORD := 16#0030;
	MIO_MODE_UNUSED:        DWORD := 16#0800;       (* Channel is not used *)

	(* Constants used as Channel-Mode for Analog-Inputs *)
	Mio_MODE_10V:			DWORD := 16#0001;		(* 16 Bits, -10V .. +10V *)
	Mio_MODE_PT100:			DWORD := 16#0002;		(* 16 Bits, temp in 1/10 Kelvin *)
	Mio_MODE_1V:			DWORD := 16#0003;		(* 16 Bits, -1V  .. +1V  *)
	Mio_MODE_20MA:			DWORD := 16#0004;		(* 16 Bits, 0mA  .. 20mA *)
	Mio_MODE_04_20MA:		DWORD := 16#0005;		(* 16 Bits, 4mA  .. 20mA *)
    Mio_MODE_PM20MA:        DWORD := 16#0006;       (* -20  ... 20mA *)
	Mio_MODE_VRangeMsk:		DWORD := 16#0007; 		(* Mask for voltage range *)
    Mio_MODE_PT100_2:       DWORD := 16#0002;       (* PT100 2 Leitertechnik *)
	Mio_MODE_PT100_3:       DWORD := 16#0020;       (* PT100 3 Leitertechnik *)
    Mio_MODE_PT1000_2:      DWORD := 16#0040;       (* PT1000 2 Leitertechnik *)
    Mio_MODE_PT1000_3:      DWORD := 16#0080;       (* PT1000 3 Leitertechnik *)
    Mio_MODE_Thermo_J:      DWORD := 16#0100;       (* Thermoelement Type J *)
    Mio_MODE_Thermo_K:      DWORD := 16#0200;       (* Thermoelement Type K *)
    Mio_MODE_Thermo_N:      DWORD := 16#0400;       (* Thermoelement Type N *)
    Mio_MODE_Thermo_S:      DWORD := 16#0800;       (* Thermoelement Type S *)
	Mio_MODE_DMS:			DWORD := 16#0008; 		(* 16 Bits, 0mV  .. 16mV *)
	Mio_MODE_SPZENT:		DWORD := 16#0009; 		(* 16 Bits, -100% .. +100% *)
	Mio_MODE_UPZENT:		DWORD := 16#000A; 		(* 16 Bits, 0%  .. 100% *)
	Mio_MODE_S5A:			DWORD := 16#000B; 		(* 16 Bits, -5A .. +5A *)
	Mio_MODE_UINT:			DWORD := 16#0100; 		(* 32 Bits, 0 .. 4294967295 *)
	Mio_MODE_SINT:			DWORD := 16#0101; 		(* 32 Bits, -2147483648 .. +2147483647 *)
	Mio_MODE_XINT:			DWORD := 16#0102; 		(* 32 Bits, Hex 0 .. 0xFFFFFFFF *)
	Mio_MODE_FREQ:			DWORD := 16#0103; 		(* 32 Bits, -262143 .. +262143 *)

	(* Constants used as Channel-Mode for AI204-Inputs *)
	(* Mio_MODE_Sync:		DWORD := 16#0008;	already defined *)
	Mio_MODE_Filt333Hz:		DWORD := 16#0000;		(* Filter with 333 Hz *)
	Mio_MODE_Filt4KHz:		DWORD := 16#0010;		(* Filter with 4 KHz *)
	Mio_MODE_Fil50Hz:       DWORD := 16#0040;       (* filter with 50 Hz *)
    Mio_MODE_Filt60Hz:      DWORD := 16#0080;       (* filter with 60 Hz *)
	Mio_MODE_NoTempComp:	DWORD := 16#0020;		(* Temperature compensation OFF *)
	Mio_MODE_Sample1:		DWORD := 16#0000;		(* 1 time sampling *)
	Mio_MODE_Sample8:		DWORD := 16#0100;		(* 8 times sampling *)
	Mio_MODE_Sample16:		DWORD := 16#0200;		(* 16 times sampling *)
	Mio_MODE_Sample32:		DWORD := 16#0300;		(* 32 times sampling *)
	Mio_MODE_SampleMsk:		DWORD := 16#0300; 		(* mask for sampling *)

	(* Constants used as Channel-Mode for ISI202 INC-Inputs/DIO2xx CNT-channels *)
	Mio_MODE_Interpol0:		DWORD := 16#0000;		(* SCI-Interpolation 0 *)
	Mio_MODE_Interpol1:		DWORD := 16#0010;		(* SCI-Interpolation 1 *)
	Mio_MODE_Interpol2:		DWORD := 16#0020;		(* SCI-Interpolation 2 *)
	Mio_MODE_Interpol3:		DWORD := 16#0030;		(* SCI-Interpolation 3 *)
	Mio_MODE_PulseDir:		DWORD := 16#0000;		(* Pulse-Direction-Mode *)
	Mio_MODE_Single:		DWORD := 16#0040;		(* 1-time counting *)
	Mio_MODE_Double:		DWORD := 16#0080;		(* 2-time counting *)
	Mio_MODE_Quad:			DWORD := 16#00C0;		(* 4-time counting *)
	Mio_MODE_Reset:			DWORD := 16#0100;		(* Activate search home *)
	Mio_MODE_NoZero:		DWORD := 16#0200;		(* Ignore encoder zero *)
	Mio_MODE_NoHome:		DWORD := 16#0400;		(* Ignore home signal *)
	Mio_MODE_AutoLd:		DWORD := 16#1000;		(* Autoreload in reference compare *)
	Mio_MODE_LatchRef:		DWORD := 16#4000;		(* Latch into reference at home *)
	Mio_MODE_LatchStrobe:	DWORD := 16#8000;		(* Latch into strobe at home *)

	(* Constants used as Channel-Mode for ISI202 SSI-Inputs *)
	Mio_MODE_Vr:			DWORD := 16#0002;		(* V/R output to high *)
	Mio_MODE_Set:			DWORD := 16#0004;		(* Set output to high *)
	Mio_MODE_NoPrty:		DWORD := 16#0000;		(* No parity *)
	Mio_MODE_Even:			DWORD := 16#0200;		(* Even parity *)
	Mio_MODE_Odd:			DWORD := 16#0400;		(* Odd parity *)
	Mio_MODE_PariMsk:       DWORD := 16#0600;       (* Mask for parity *)
	Mio_MODE_Bin:			DWORD := 16#0000;		(* Binary data format *)
	Mio_MODE_Gray:			DWORD := 16#0800;		(* Gray-Code data format *)

	(* Constants used as Channel-Mode for ISI202/DIO2xx CNT-channels *)
	Mio_MODE_Inc:			DWORD := 16#0000;		(* Incremental mode *)
	Mio_MODE_Ssi:			DWORD := 16#0001;		(* Synchronous serial mode *)
	Mio_MODE_Sync:			DWORD := 16#0008;		(* no effect in SSI-Mode *)
	MIO_M_LATHOME_R:        DWORD := 16#00004000;   (* Latch into reference at home *)
	MIO_M_LATHOME_S:  		DWORD := 16#00008000;  	(* Latch into strobe at home *)
    MIO_M_LATTRIG_S:        DWORD := 16#00010000;   (* Latch into trig at home *)
	Mio_MODE_Continuous:    DWORD := 16#00020000;   (* Continuous homing *)
	MIO_M_GATETIME:     	DWORD := 16#00100000;   (* Measure gatetime *)
	MIO_M_PERIOD:       	DWORD := 16#00200000;   (* Measure period *)
	MIO_M_AUTO:             DWORD := 16#00300000;   (* Auto. determine GATE or PERIOD *)

	(* Constants used as Card-Mode for ISI202  *)
	Mio_MODE_FastPFail:		DWORD := 16#2000;		(* Fast Power-Fail enable *)

	(* Constants used as Channel-Mode for CNT204/DIO2xx CNT-channels *)
	(* Mio_MODE_Inc:		DWORD := 16#0000;	only channel 1 and 2 *)
	Mio_MODE_Count:			DWORD := 16#0002;	(* Counter mode *)
	Mio_MODE_Trigg:			DWORD := 16#0003;	(* only channel 3 and 4 *)
	MIO_M_PULSEDIR:  	    DWORD := 16#00000000;   (* Pulse-Direction-Mode *)
	(* Already defined for ISI *)
	(* Mio_MODE_Sync:		DWORD := 16#0008;	already defined *)
	(* Mio_MODE_PulseDir:	DWORD := 16#0000;	only in INC-Mode *)
	(* Mio_MODE_Single:		DWORD := 16#0040;	only in INC-Mode *)
	(* Mio_MODE_Double:		DWORD := 16#0080;	only in INC-Mode *)
	(* Mio_MODE_Quad:		DWORD := 16#00C0;	only in INC-Mode *)
	(* Mio_MODE_Reset:		DWORD := 16#0100; *)
	(* Mio_MODE_NoZero:		DWORD := 16#0200;	only in INC-Mode *)
	(* Mio_MODE_NoHome:		DWORD := 16#0400;	only in INC-Mode *)

	Mio_MODE_CntTime:		DWORD := 16#0800;	(* Measure time between counts *)
	Mio_MODE_IncTime:		DWORD := 16#1000;	(* Measure time between increments *)
	Mio_MODE_DiffTime:		DWORD := 16#2000;	(* Measure time difference  *)

	(* Constants used as Channel-Modes for DMS202 *)
	Mio_MODE_2MV:			DWORD := 16#0001;	(* Input range is 2mV *)
	Mio_MODE_4MV:			DWORD := 16#0002;	(* Input range is 4mV *)
	Mio_MODE_8MV:			DWORD := 16#0004;	(* Input range is 8mV *)
	Mio_MODE_16MV:			DWORD := 16#0008;	(* Input range is 16mV *)
	Mio_MODE_AutoR:			DWORD := 16#000F;	(* Auto Range *)
	Mio_MODE_DmsRanMsk:		DWORD := 16#000F; 	(* Mask for DMS range *)
	Mio_MODE_IncModMsk:		DWORD := 16#00C0; 	(* Mask for INC mode *)

	(* Possible values for MIO_SETCHMOD_C.Mode AND MIO_GETCHMOD_C.Mode *)
	(* in CASE OF a PWM202 *)
    Mio_MODE_Brake:			DWORD := 16#0000;	(* PWM brake on *)
    Mio_MODE_Operate:		DWORD := 16#0001;	(* PWM running  *)
    Mio_MODE_RunMsk:		DWORD := 16#0001;	(* Mask for PWM modes operate *)

    Mio_MODE_Pwm:			DWORD := 16#0000;	(* SMA/LAP PWM-control is active *)
    Mio_MODE_Control:		DWORD := 16#0002;	(* SMA/LAP I-control is active *)
    Mio_MODE_ContMsk:		DWORD := 16#0002;	(* Mask for PWM- OR I-control *)

	Mio_MODE_ResLo:         DWORD := 16#0000;   (* 5.0 A AD-converter resolution *)
	Mio_MODE_ResHi:         DWORD := 16#0004;   (* 1.5 A AD-Converter resolution *)
	Mio_MODE_ResMsk:        DWORD := 16#0004;   (* Resolution mask *)

    Mio_MODE_Sma:			DWORD := 16#0000;	(* Sign/Magnitude control setting *)
    Mio_MODE_Lap:			DWORD := 16#0008;	(* Locked antiphase control setting *)
    Mio_MODE_ModeMsk:		DWORD := 16#0008;	(* Mask for PWM- OR I-control *)

    Mio_MODE_Open:			DWORD := 16#0000;	(* no shorting open switches*)
    Mio_MODE_Upper:			DWORD := 16#0010;	(* shorting using upper switches *)
    Mio_MODE_Lower:			DWORD := 16#0020;	(* shorting using lower switches *)
    Mio_MODE_BrakeMsk:		DWORD := 16#0030;	(* Mask for PWM modes brakes *)

    Mio_MODE_Edge:			DWORD := 16#0000;	(* Pulse width switch align edge *)
    Mio_MODE_Center:		DWORD := 16#0040;	(* Pulse width switch align center *)
    Mio_MODE_AlignMsk:		DWORD := 16#0040;	(* Mask for PWM mode others *)

    Mio_MODE_PreScal:		DWORD := 16#0080;	(* 256us prescale active NOT app. *)
    Mio_MODE_PreScMsk:		DWORD := 16#0080;	(* Mask for prescale *)

    Mio_MODE_PwmUsrMsk:		DWORD := 16#007B;
	(* MIO_M_ALIGNMSK | MIO_M_BRAKEMSK | MIO_M_MODEMSK |
 	   MIO_M_CONTMSK | MIO_M_RUNMSK *)

    (* Possible values for MIO_SETCHMOD_C.Mode AND MIO_GETCHMOD_C.Mode *)
    (* in CASE OF a SLC284, SDO204, SDI208 *)
    MIO_M_SAFETY_ERROR:           DWORD := 16#00000001;  (* Safety module in error status *)
    MIO_M_SAFETY_PROG:            DWORD := 16#00000002;  (* Safety module in programming mode *)
    MIO_M_SAFETY_TEST:            DWORD := 16#00000004;  (* Safety module in test mode *)
    MIO_M_SAFETY_SAFE:            DWORD := 16#00000008;  (* Safety module in safe mode *)
    MIO_M_SAFETY_WAITFORSAFE:     DWORD := 16#00000010;  (* Safety module waiting for safe mode *)
    MIO_M_SAFETY_BIOS:            DWORD := 16#00000020;  (* Safety module only Bios active *)
	MIO_M_SAFETY_SAFEDELAY:       DWORD := 16#00000040;  (* Safety module in safe delay mode *)
	MIO_M_SAFETY_GOLDEN_REF:      DWORD := 16#00000080;  (* Safety module in golden reference mode (FPGA only) *)

	(* in case of a PVA2XX *)

	MIO_M_PVA_UNIPOLAR:         DWORD := 16#0001;   (* Half-Bridge *)
	MIO_M_PVA_BIPOLAR:          DWORD := 16#0002;   (* H-Bridge *)
	MIO_M_PVA_UNIPOLAR2COIL:    DWORD := 16#0004;   (* Unipolar with 2 coils *)
	MIO_M_PVA_UNUSED:           DWORD := 16#0800;   (* Channel is not used *)
	MIO_M_PVA_DISABLED:         DWORD := 16#1000;   (* Channel is deactivated *)
	MIO_M_PVA_ENABLED:          DWORD := 16#2000;   (* Channel is activated *)

	(* GIO2xx *)
	(*--- Module modes ---*)
	MIO_M_GIORUN:   			  DWORD := 16#00000001;   (* Run mode of the module *)
	MIO_M_GIOSTOP:  			  DWORD := 16#00000002;   (* Stop mode *)
	(* Specific modes for digital inputs and counters *)
	MIO_M_GIOSPECDITYPE3:         DWORD := 16#00000000;  (* Digital input type 3 *)
	MIO_M_GIOSPECDITYPE2:         DWORD := 16#00000200;  (* Digital input type 2 *)
	MIO_M_GIOSPECDITYPE1:         DWORD := 16#00000400;  (* Digital input type 1 *)
	MIO_M_GIOSPECDISOURCE:        DWORD := 16#00000600;  (* Digital input type source *)
	MIO_M_GIOSPECDICMP:           DWORD := 16#00000800;  (* Digital input type comparator *)
	MIO_M_GIOSPECDIMODES:         DWORD := 16#00000E00;  (* Special modes for digital inputs *)
    (* Global channel modes *)
	MIO_M_GIODISABLED:            DWORD := 16#00000000;  (* Channel is disabled *)
	MIO_M_GIODISOURCE:            DWORD := 16#00000610;  (* Digital input pull-up *)
	MIO_M_GIODITYPE1:             DWORD := 16#00000410;  (* Digital input type 1 *)
	MIO_M_GIODITYPE2:             DWORD := 16#00000210;  (* Digital input type 2 *)
	MIO_M_GIODITYPE3:             DWORD := 16#00000010;  (* Digital input type 3 *)
	MIO_M_GIODITYPECMP:           DWORD := 16#00000810;  (* Digital input type comparator *)
	MIO_M_GIODOPUSHPULL:          DWORD := 16#00000021;  (* Digital output push pull *)
	MIO_M_GIODOIOLINK:            DWORD := 16#00000022;  (* IO-Link (set only per configuration) *)
	MIO_M_GIODOLOWSIDE:           DWORD := 16#00000023;  (* Digital output low-side driver *)
	MIO_M_GIODOHIGHSIDE:          DWORD := 16#00000024;  (* Digital output high-side driver *)
	MIO_M_GIOVI_10V:              DWORD := 16#00000031;  (* Voltage input -10V..10V *)
	MIO_M_GIOVI_1V:               DWORD := 16#00000032;  (* Voltage input -1V..1V *)
	MIO_M_GIOVI_100mV:            DWORD := 16#00000033;  (* Voltage input -100mV..100mV *)
	MIO_M_GIOVI_10mV:             DWORD := 16#00000034;  (* Voltage input -10mV..10mV *)
	MIO_M_GIOVIRANGE1:            DWORD := 16#00000035;  (* Voltage input -17.5mV..87.5mV *)
	MIO_M_GIOVIRANGE2:            DWORD := 16#00000036;  (* Voltage input -4.375mV..21.875mV *)
	MIO_M_GIOVO:                  DWORD := 16#00000041;  (* Voltage output -10V..10V *)
	MIO_M_GIOVOEXT:               DWORD := 16#00000042;  (* Extended voltage output (supply for sensors) *)
	MIO_M_GIOCI_20mA:             DWORD := 16#00000051;  (* Current input -20mA..20mA *)
	MIO_M_GIOCI_4_20mA:           DWORD := 16#00000052;  (* Current input 4mA..20mA *)
    MIO_M_GIOCI_0_20mA:           DWORD := 16#00000053;  (* Current input 0mA..20mA *)
	MIO_M_GIOCO_0_20mA:           DWORD := 16#00000061;  (* Current output 0mA..20mA *)
	MIO_M_GIOCO_4_20mA:           DWORD := 16#00000062;  (* Current output 4mA..20mA *)
	MIO_M_GIOCO_0_2mA:            DWORD := 16#00000063;  (* Current output 0mA..2mA *)
	MIO_M_GIOCO_0_200uA:          DWORD := 16#00000064;  (* Current output 0uA..200uA *)
	MIO_M_GIOCNTEDGE:             DWORD := 16#00000091;  (* Counter - Edge *)
	MIO_M_GIOCNTTIMEPERIOD:       DWORD := 16#00000092;  (* Counter - Time period *)
	MIO_M_GIOCNTTIMEPULSE:        DWORD := 16#00000093;  (* Counter - Time pulse *)
	MIO_M_GIOCNTDUALEDGETRIG:     DWORD := 16#000000A1;
	MIO_M_GIOCNTDUALEDGERESET:    DWORD := 16#000000A2;
	MIO_M_GIOCNTDUALEDGEGATE:     DWORD := 16#000000A3;
	MIO_M_GIOCNTDUALEDGEDIR:      DWORD := 16#000000A4;
	MIO_M_GIOCNTDUALEDGETIME:     DWORD := 16#000000A5;
	MIO_M_GIOCNTINC_1:            DWORD := 16#000000B1;
	MIO_M_GIOCNTINC_2:            DWORD := 16#000000B2;
	MIO_M_GIOCNTINC_4:            DWORD := 16#000000B3;
	MIO_M_GIOPWMPUSHPULL:         DWORD := 16#00000071;  (* Pulse width modulation - push pull *)
	MIO_M_GIOPWMLOWSIDE:          DWORD := 16#00000073;  (* Pulse width modulation - low-side driver *)
	MIO_M_GIOPWMHIGHSIDE:         DWORD := 16#00000074;  (* Pulse width modulation - high-side driver *)
	MIO_M_GIOPWMDUALPUSHPULL:     DWORD := 16#00000081;  (* Pulse width modulation with second channel - push pull *)
	MIO_M_GIOPWMDUALLOWSIDE:      DWORD := 16#00000083;  (* Pulse width modulation with second channel - low-side driver *)
	MIO_M_GIOPWMDUALHIGHSIDE:     DWORD := 16#00000084;  (* Pulse width modulation with second channel - high-side driver *)
	MIO_M_GIOTEMOELEM_J:          DWORD := 16#000000C1;  (* Termo element type J *)
	MIO_M_GIOTEMOELEM_K:          DWORD := 16#000000C2;  (* Termo element type K *)
	MIO_M_GIOTEMOELEM_T:          DWORD := 16#000000C3;  (* Termo element type T *)
	MIO_M_GIOTEMOELEM_N:          DWORD := 16#000000C4;  (* Termo element type N *)
	MIO_M_GIOTEMOELEM_E:          DWORD := 16#000000C5;  (* Termo element type E *)
	MIO_M_GIOTEMOELEM_R:          DWORD := 16#000000C6;  (* Termo element type R *)
	MIO_M_GIOTEMOELEM_S:          DWORD := 16#000000C7;  (* Termo element type S *)
	MIO_M_GIOTEMOELEM_B:          DWORD := 16#000000C8;  (* Termo element type B *)
	MIO_M_GIOPT100_2:             DWORD := 16#000000D1;  (* Temperature sensor of type PT100 - 2 wire *)
	MIO_M_GIOPT100_3:             DWORD := 16#000000D2;  (* Temperature sensor of type PT100 - 3 wire *)
	MIO_M_GIOPT100_4:             DWORD := 16#000000D3;  (* Temperature sensor of type PT100 - 4 wire *)
	MIO_M_GIOPT200_2:             DWORD := 16#000000D4;  (* Temperature sensor of type PT200 - 2 wire *)
	MIO_M_GIOPT200_3:             DWORD := 16#000000D5;  (* Temperature sensor of type PT200 - 3 wire *)
	MIO_M_GIOPT200_4:             DWORD := 16#000000D6;  (* Temperature sensor of type PT200 - 4 wire *)
	MIO_M_GIOPT500_2:             DWORD := 16#000000D7;  (* Temperature sensor of type PT500 - 2 wire *)
	MIO_M_GIOPT500_3:             DWORD := 16#000000D8;  (* Temperature sensor of type PT500 - 3 wire *)
	MIO_M_GIOPT500_4:             DWORD := 16#000000D9;  (* Temperature sensor of type PT500 - 4 wire *)
	MIO_M_GIOPT1000_2:            DWORD := 16#000000DA;  (* Temperature sensor of type PT1000 - 2 wire *)
	MIO_M_GIOPT1000_3:            DWORD := 16#000000DB;  (* Temperature sensor of type PT1000 - 3 wire *)
	MIO_M_GIOPT1000_4:            DWORD := 16#000000DC;  (* Temperature sensor of type PT1000 - 4 wire *)
	MIO_M_GIOIOLINK:              DWORD := 16#000000E0;  (* IO Link *)
	MIO_M_GIODODUALPUSHPULL:      DWORD := 16#000000f1;  (* Digital output with second channel - push pull *)
	MIO_M_GIODODUALLOWSIDE:       DWORD := 16#000000F3;  (* Digital output with second channel - low-side driver *)
	MIO_M_GIODODUALHIGHSIDE:      DWORD := 16#000000F4;  (* Digital output with second channel - high-side driver *)
	MIO_M_GIOFRQHIGHSIDE:         DWORD := 16#00000114;   (* Frequency modulation push pull *)
    MIO_M_GIOFRQPUSHPULL:         DWORD := 16#00000111;   (* Frequency modulation low side *)
	MIO_M_GIOFRQLOWSIDE:          DWORD := 16#00000113;   (* Frequency modulation high side *)
    (* Additional channel modes invert *)
	MIO_M_GIOINVERT:              DWORD := 16#00001000;  (* Invert the value *)
    (* Combined channel modes *)
	MIO_M_GIOPUSHPULL:            DWORD := 16#00000000;  (* Inverted signal AT combined outputs *)
	MIO_M_GIOPUSHPUSH:            DWORD := 16#00002000;  (* Same output signal at combined channels *)
    (* Additional channel modes - digital *)
	MIO_M_GIOFAST:                DWORD := 16#00004000;  (* Inputs/Outputs: use fast input/output *)
	MIO_M_GIODOPULSE:             DWORD := 16#00008000;  (* Output only: use PWM to reduce output current *)
    (* Additional channel modes - edge counter *)
	MIO_M_GIOCNTUP:               DWORD := 16#00000000;  (* Count up *)
	MIO_M_GIOCNTDOWN:             DWORD := 16#00010000;  (* Count down *)
	MIO_M_GIORISING:              DWORD := 16#00020000;  (* Count rising edges *)
	MIO_M_GIOFALLING:             DWORD := 16#00040000;  (* Count falling edges *)
	MIO_M_GIOBOTH:                DWORD := 16#00060000;  (* Count both edges *)
	MIO_M_RESETATREFERENCE:       DWORD := 16#00080000;  (* Reset at reference *)
    (* Additional channel modes - PWM *)
    MIO_M_GIOPWMNOTLOCKED:        DWORD := 16#00000000;   (* Simple PWM (not in locked antiphase mode) *)
	MIO_M_GIOPWMLOCKED:			  DWORD := 16#00100000;   (* PWM in locked antiphase mode *)
    (* Additional channel modes - General *)
	MIO_M_GIOSYNC:                DWORD := 16#00200000;   (* Use Sync for channel *)
	MIO_M_GIOLIMITERROR:          DWORD := 16#00800000;   (* Use limits as error *)
	MIO_M_GIOFIFO:                DWORD := 16#01000000;   (* Use FIFO for measurement *)
	MIO_M_GIOFREQUENCY:           DWORD := 16#02000000;   (* Frequency modulation *)
	MIO_M_GIOPULSE:               DWORD := 16#04000000;   (* Pulse modulation *)
	(*--- Additional channel modes - Thermo couples ---*)
	MIO_M_GIOGROUNDED: 			  DWORD := 16#00400000;   (* Use grounded junction probe *)
    (*--- Special mode for CAN ---*)
	MIO_M_GIOCANCONFIG:           DWORD := 16#80000000;   (* Stop card before setting channel mode and start card again - only for CAN! *)

	(* Possible commands for all IO modules *)
	Mio_CMD_GetVersion:		DINT := 50;			(* Get driver AND firmware version *)
    Mio_CMD_GetErrStatist:  DINT := 54;         (* Get module error statistics *)

	(* CCM202, ACR222, DPM200 *)
	Mio_CMD_UpdateSw:		DINT := 9; 			(* Update firmware on module *)

	(* FM2xx, FS2xx *)
	Mio_CMD_TrigWDog:		DINT := 30; 		(* Trigger watchdog *)
	Mio_CMD_ClrInt:			DINT := 31; 		(* Clear event interrupt *)

	(* DPM200 *)
	Mio_CMD_SetParameter:	DINT := 40; 		(* Set network parameters *)
	Mio_CMD_SetMode:		DINT := 41; 		(* Set mode for user interface *)
	Mio_CMD_GetMode:		DINT := 42; 		(* Set mode on user interface *)
	Mio_CMD_Mark:			DINT := 43; 		(* Wait for token *)
	Mio_CMD_LoadBusPar:		DINT := 44; 		(* Load bus parameters *)
	Mio_CMD_ReadBusPar:		DINT := 45; 		(* Read bus parameters *)
	Mio_CMD_GlobalCtrl:		DINT := 46; 		(* New mode for slave(s) *)
	Mio_CMD_SetRawParam:	DINT := 47; 		(* Set network parameters per file *)

	(* AI204 *)
	Mio_CMD_TempComp:		DINT := 60; 		(* Start temperature compensation *)
	Mio_CMD_ReadCalib:      DINT := 61;    		(* Read Calibration Data *)
	Mio_CMD_GetEvent:       DINT := 62;    		(* Read event flags *)

    (* AI208/SI *)
	Mio_CMD_SetMinMaxEvent: DINT := 63;			(* Set event configuration *)
	Mio_CMD_GetMinMaxEvent: DINT := 64;			(* Get event configuration *)
	Mio_CMD_SetMinMaxError: DINT := 65;			(* Set error configuration *)
	Mio_CMD_GetMinMaxError: DINT := 66;			(* Get error configuration *)

	(* Constants used as Command-Code (Mio_DoCmd()) with INC- or COUNT-Inputs *)
	Mio_CMD_SetRef:			DINT := 1;			(* only in INC-Mode *)
	Mio_CMD_ZInit:			DINT := 5;			(* only in INC-Mode *)
	Mio_CMD_GetRst:			DINT := 7;			(* only in INC-Mode/Read search home status *)
	Mio_CMD_EnableRst:		DINT := 12;			(* only in INC-Mode/Activate search home *)
	Mio_CMD_DisableRst:		DINT := 13;			(* only in INC-Mode/De-activate search home *)
	Mio_CMD_GetStrobe:		DINT := 21;			(* only in INC-Mode/Get strobe register value *)
	Mio_CMD_GetRef:			DINT := 22;			(* only in INC-Mode *)
	Mio_CMD_GetAct:			DINT := 23;			(* only on CNT204 *)
	Mio_CMD_GetStrbStat:	DINT := 24;			(* only in INC-Mode on CNT204 *)
	Mio_CMD_GetInpStat:		DINT := 25;			(* only on CNT204 *)
	Mio_CMD_GetZeroStat:	DINT := 26;			(* only in INC-Mode on CNT204 *)

	(* Constants used as Command-Code (Mio_DoCmd()) with SSI-Inputs *)
	Mio_CMD_SetFreq:		DINT := 2;
	Mio_CMD_SetDLen:		DINT := 3;
	Mio_CMD_SetInterval:	DINT := 6;

	(* Constants used as Command-Code (Mio_DoCmd()) with ISI202-Card *)
	Mio_CMD_Reset:			DINT := 4;
	Mio_CMD_SetFilter:		DINT := 20;      (* Set filter frequency *)
    Mio_CMD_GetFrequency:   DINT := 27;      (* Get internal frequency *)
	MIO_CMD_GETFREQ:        DINT := 143;
	MIO_CMD_GETINTERVAL:    DINT := 144;
	MIO_CMD_GETDLEN:        DINT := 145;
	MIO_CMD_GETRESETVALUE:  DINT := 146;
	Mio_CMD_SetResetvalue:	DINT := 147;
	MIO_CMD_SIMERROR:       DINT := 148;
	MIO_CMD_SIMEVENT:       DINT := 149;
	MIO_CMD_SETACTIVE:      DINT := 150;
	MIO_CMD_GETENCRES:      DINT := 151;
	MIO_CMD_SETENCRES:      DINT := 152;
	MIO_CMD_GETGATETIME:    DINT := 153;
	MIO_CMD_SETGATETIME:    DINT := 154;
	MIO_CMD_GETDISTANCEREF: DINT := 155;
	MIO_CMD_SETDISTANCEREF: DINT := 156;
	MIO_CMD_CONFIGNULLEDGE: DINT := 157;
	MIO_CMD_GETNULLEDGE:    DINT := 158;
	MIO_CMD_ENABLENULL:     DINT := 159;
	MIO_CMD_ISNULLENABLED:  DINT := 160;
	MIO_CMD_ISRESETPENDING: DINT := 161;
	MIO_CMD_GETACTIVELEVEL: DINT := 162;
	MIO_CMD_SETACTIVELEVEL: DINT := 163;
	MIO_CMD_SETTESTMODE:    DINT := 164;

	(* Constants used as parameters for MIO_CMD_GETACTIVELEVEL *)
	MIO_HIGHACTIVE: DWORD := 16#0001;
	MIO_LOWACTIVE:  DWORD := 16#0002;


	(* Constants used as Command-Code (Mio_DoCmd()) with DMS202-Card *)
	Mio_CMD_PeekRw:			DINT := 1000;		(* Read and reset peek value *)
	Mio_CMD_PeekRo:			DINT := 1001;		(* Read peek value *)
	Mio_CMD_ZeroCalib:		DINT := 1027;		(* Calibration with C + O *)
	Mio_CMD_ZeroCalibTmp:	DINT := 1039;		(* Temporary calibration with C + O *)
	Mio_CMD_OffsetCal:		DINT := 1028;		(* Calibration only with O *)
	Mio_CMD_OffsetCalTmp:	DINT := 1040;		(* Temporary calibration only with O *)

	(* Constants used as Command-Code (Mio_DoCmd4()) with ACR222-Card *)
	Mio_CMD_GetVal:			DINT := 10;			(* Read specific value *)
	Mio_CMD_SetVal:			DINT := 11;			(* Write specific value *)
	Mio_CMD_GetActVal:		DINT := 14; 		(* Read actual value *)
	Mio_CMD_GetSetVal:		DINT := 15; 		(* Write set value *)
	Mio_CMD_GetNewSet:		DINT := 16; 		(* Conditional read *)

    (* Constants used as Command-Code with ACR222-Card in Channel Mode *)
    Mio_CMD_SetProf:       		DINT := 17;     		(* Set Profile *)
	Mio_CMD_GetProf:       		DINT := 18;     		(* Get Profile *)
	Mio_CMD_SetQuickDecel: 		DINT := 19;     		(* Set Quick Deceleration *)
	Mio_CMD_GetQuickDecel: 		DINT := 20;     		(* Get Quick Deceleration *)
	Mio_CMD_SetHome:	   		DINT := 21;     		(* Set Home Parameters *)
	Mio_CMD_GetHome:	   		DINT := 22;          	(* Get Home Parameters *)
	Mio_CMD_SetCommonSettings: 	DINT := 23;   		 	(* Set Common Settings *)
	Mio_CMD_GetCommonSettings:  DINT := 24;			    (* Get Common Settings *)
	Mio_CMD_SetDriveData:	    DINT := 27;		     	(* Set Drive Data *)
    Mio_CMD_GetDriveData:	    DINT := 28;		      	(* Get Drive Data *)
    Mio_CMD_SetResolution: 		DINT := 29;		        (* Set Resolution *)
	Mio_CMD_GetResolution: 		DINT := 30;		        (* Get Resolution *)
    Mio_CMD_SetErrorWindow: 	DINT := 31;  	    	(* Set Error Window *)
    Mio_CMD_GetErrorWindow: 	DINT := 32;      		(* Get Error Window *)
	Mio_CMD_SetMaxFreq: 	 	DINT := 33;		        (* Set Maximum Frequency *)
    Mio_CMD_GetMaxFreq:			DINT := 34;		        (* Set Maximum Frequency *)

	Mio_CMD_GetSwitchState: 	DINT := 35;
    Mio_CMD_GetStateHist: 		DINT := 36;
    Mio_CMD_SwitchToChannels: 	DINT := 37;

	(* Possible commands for the IO module PWM202 *)
    Mio_CMD_SetPP:			DINT := 70;	  (* Set puls period duration uS *)
    Mio_CMD_GetPP:			DINT := 71;	  (* Get puls period duration uS *)
    Mio_CMD_SetOP:			DINT := 72;	  (* Set operation mode on/off *)
    Mio_CMD_GetOP:			DINT := 73;	  (* Get operation mode *)
    Mio_CMD_GetTemp:		DINT := 74;	  (* Get actual card temperature *)
    Mio_CMD_SetPar_Base:	DINT := 80;
    Mio_CMD_SetPar_Ts:		DINT := 80;	  (* Set controler sample TIME *)
    Mio_CMD_SetPar_Pr:		DINT := 81;	  (* Set controler proportional range *)
    Mio_CMD_SetPar_Ti:		DINT := 82;   (* Set controler integration TIME *)
    Mio_CMD_SetPar_Td:		DINT := 83;   (* Set controler differentation TIME *)
    Mio_CMD_GetPar_Base:	DINT := 90;
    Mio_CMD_GetPar_Ts:		DINT := 90;	  (* Get controler sample TIME *)
    Mio_CMD_GetPar_Pr:		DINT := 91;   (* Get controler proportional range *)
    Mio_CMD_GetPar_Ti:		DINT := 92;	  (* Get controler integration TIME *)
    Mio_CMD_GetPar_TD:		DINT := 93;	  (* Get controler differentation TIME *)
	Mio_CMD_MaxCurrent:     DINT  := 100; (* Maximum current *)
	Mio_CMD_CurrentRes:     DINT  := 101; (* Current resolution *)
	Mio_CMD_LoadType:       DINT  := 102; (* Set load current *)
	Mio_CMD_GetMaxCurrent:  DINT  := 103; (* Get maximum current *)
	Mio_CMD_GetLoadType:    DINT  := 104; (* Get load current *)
	Mio_CMD_GetCurrentRes:  DINT  := 105; (* Get current resolution *)

	(* Possible commands for the IO module CNT204 with TIME mode support *)
	Mio_CMD_LostTimeVal:	DINT := 120; (* Query IF a value has been lost *)
	Mio_CMD_NewTimeVal:		DINT := 121; (* Query if a new value is available *)

    (* Possible commands for the IO module DIO2xx *)
    Mio_CMD_GetFilter:      DINT := 140;  (* Read filter configuration *)
    MIO_CMD_GETPWMCFG:      DINT := 420;  (* Read PWM configuration OF DO channel *)
    MIO_CMD_SETPWMCFG:      DINT := 421;  (* Write PWM configuration OF DO channel *)
	MIO_CMD_GETPINLEVELS:   DINT := 422;  (* Read pin levels of DIO channels *)

	(* Possible commands for the driver ECAT201 *)
	MIO_CMD_DCRESET:            DINT  := 170;   (* Obsolete *)
	MIO_CMD_STOPMASTER:         DINT  := 171;   (* Stop EtherCAT master *)
	MIO_CMD_STARTMASTER:        DINT  := 172;   (* Start EtherCAT master *)
	MIO_CMD_RAWCMD:             DINT  := 173;   (* Send raw EtherCAT command *)
	MIO_CMD_SDOREAD:            DINT  := 174;   (* Read SDO (CoE) *)
	MIO_CMD_SDOWRITE:           DINT  := 175;   (* Write SDO (CoE) *)
	MIO_CMD_GETOBJDICT:         DINT  := 176;   (* Get object dictionary (CoE) *)
	MIO_CMD_GETOBJDESC:         DINT  := 177;   (* Get object description (CoE) *)
	MIO_CMD_GETOBJENTRY:        DINT  := 178;   (* Get object entry (CoE) *)
	MIO_CMD_GETEMCY:            DINT  := 179;   (* Get emergency (CoE) *)
	MIO_CMD_GETMASTERSTATE:     DINT  := 180;   (* Get master state *)
	MIO_CMD_SETMASTERSTATE:     DINT  := 181;   (* Set master state *)
	MIO_CMD_GETSLAVESTATE:      DINT  := 182;   (* Get slave state *)
	MIO_CMD_SETSLAVESTATE:      DINT  := 183;   (* Set slave state *)
	MIO_CMD_SETDATAVALID:       DINT  := 184;   (* Set data valid now (DMW200) *)
	MIO_CMD_GETCYCLEERROR:      DINT  := 185;   (* Get cycle error (DMW200) *)
	MIO_CMD_RESETCYCLEERROR:    DINT  := 186;   (* Reset cycle error (DMW200) *)
	MIO_CMD_GETCYCLETIME:       DINT  := 187;   (* Get cycle time configuration (DMW200) *)
	MIO_CMD_EXCLUDESLAVE:       DINT  := 188;   (* Exclude slave from configuration *)
	MIO_CMD_GETALIASADDR:       DINT  := 189;   (* Get slave alias address *)
	MIO_CMD_SETALIASADDR:       DINT  := 190;   (* Set slave alias address *)
	MIO_CMD_FILEWRITE:          DINT  := 192;   (* Write file (FoE) *)
	MIO_CMD_SERVOREAD:          DINT  := 193;   (* Read SoE value *)
	MIO_CMD_SERVOWRITE:         DINT  := 194;   (* Write SoE value *)

    (* Possible commands for the IO module AIC212 *)
	Mio_CMD_ExportValues:        DINT := 200;
	Mio_CMD_SimulateValues:      DINT := 201;
	Mio_CMD_Start:               DINT := 202;
	Mio_CMD_Stop:                DINT := 203;
	Mio_CMD_SetTempDir:          DINT := 204;
	Mio_CMD_GetTempDir:          DINT := 205;
	Mio_CMD_SetCompression:      DINT := 206;
	Mio_CMD_GetCompression:      DINT := 207;
	Mio_CMD_SetRecordLen:        DINT := 208;
	Mio_CMD_GetRecordLen:        DINT := 209;
	Mio_CMD_GetStatus:           DINT := 210;
	Mio_CMD_GetValues:           DINT := 211;
	Mio_CMD_Open:                DINT := 212;
	Mio_CMD_Close:               DINT := 213;
	Mio_CMD_ReadSamples:         DINT := 214;
	Mio_CMD_ReadHeader:          DINT := 215;
	Mio_CMD_GetMemSize:          DINT := 216;

    (* Possible commands for the IO module DOR206 *)
	Mio_CMD_GETSWITCHCOUNT:      DINT := 264;
	Mio_CMD_RESETSWITCHCOUNT:    DINT := 265;

	(* Possible command for the PN module *)
	Mio_CMD_GetErrStat:			 DINT := 302; (* Read error statistic *)
	Mio_CMD_ResetErrStat:		 DINT := 303; (* Reset error statistic *)

    (* Possible commands for the IO module SEM201 *)
    Mio_CMD_GetSetValueList:     DINT := 2001; (* Get list OF configured setvalues *)
    Mio_CMD_GetActValueList:     DINT := 2002; (* Get list of configured actvalues *)
    Mio_CMD_GetTransPower:       DINT := 2003; (* Get optical transmission power *)
    Mio_CMD_SetComPhase:         DINT := 2004; (* Set requested comm. phase *)
    Mio_CMD_GetComPhase:         DINT := 2005; (* Get current communication phase *)
    Mio_CMD_GetBaudrate:         DINT := 2006; (* Get SERCOS baudrate *)
	Mio_CMD_GetTiming:           DINT := 2007; (* Get SERCOS timings *)
    Mio_CMD_GetServiceChan:      DINT := 2009; (* Get value(S) using servicechannel *)
    Mio_CMD_SetServiceChan:      DINT := 2010; (* Set value(s) using servicechannel *)
    Mio_CMD_GetAttribute:        DINT := 2011; (* Get Attribute of IDN *)
    Mio_CMD_GetErrorMsg:         DINT := 2012; (* Get text of SERCOS error-code *)
    Mio_CMD_GetControlWord:      DINT := 2013; (* Get content OF the control WORD *)
    Mio_CMD_SetControlWord:      DINT := 2014; (* Get content of the control word *)
    Mio_CMD_GetStatusWord:       DINT := 2015; (* Get content OF the status WORD *)
    Mio_CMD_GetCmdStatus:        DINT := 2016; (* Get status OF command FUNCTION *)
    Mio_CMD_SetChanValid:        DINT := 2018; (* Confirm (validation of chan. values) *)
    Mio_CMD_GetErrCounter:       DINT := 2019; (* Get consistence error counter *)
    Mio_CMD_ResetErrCounter:     DINT := 2020; (* consistence error counter *)

    Mio_CMD_Get_Async_Sc:        DINT := 2021; (* Get value(S) using async. servicech. *)
    Mio_CMD_Set_Async_Sc:        DINT := 2022; (* Set value(S) using async. servicech. *)

	(* Possible commands for the driver MBM201 *)
	MIO_CMD_SENDMBMESSAGE:		 DINT := 3001;
	MIO_CMD_CHANGEPOLLRATE:		 DINT := 3002;
	MIO_CMD_GETPOLLRATE:		 DINT := 3003;

    (* Possible commands for safety drivers *)
    MIO_CMD_SAFETYSENDSTR:        DINT := 6001;    (* Send String *)
    MIO_CMD_SAFETYRECVSTR:        DINT := 6002;    (* Receive String *)
    MIO_CMD_SAFETYSENDBIN:        DINT := 6003;    (* Send Binary *)
    MIO_CMD_SAFETYRECVBIN:        DINT := 6004;    (* Receive Binary *)
    MIO_CMD_SAFETYSENDCMD:        DINT := 6005;    (* Send Command *)
    MIO_CMD_SAFETYSENDFILE:       DINT := 6006;    (* Send File *)
    MIO_CMD_SAFETYRECVFILE:       DINT := 6007;    (* Receive File *)
    MIO_CMD_SAFETYFILESTAT:       DINT := 6008;    (* Get file statistic *)
    MIO_CMD_SAFETYSENDRECVBIN:    DINT := 6009;    (* Send and receive binary *)
    MIO_CMD_SAFETYUSERLOGIN:      DINT := 6010;    (* User Login *)
    MIO_CMD_SAFETYUSERLOGOUT:     DINT := 6011;    (* User Logout *)
    MIO_CMD_SAFETYUSERSHOWACT:    DINT := 6012;    (* Show actual user *)
    MIO_CMD_SAFETYDOWNLOADNEWPRO: DINT := 6013;    (* Download a new SLC program *)
    MIO_CMD_SAFETYGETUID:         DINT := 6014;    (* get unique ID of SLC *)
    MIO_CMD_SAFETYASSIGNMODULES:  DINT := 6015;    (* assign modules *)
    MIO_CMD_SAFETYDBGRUN:         DINT := 6016;    (* Run in debug mode *)
    MIO_CMD_SAFETYDBGSTOP:        DINT := 6017;    (* Stop in debug mode *)
    MIO_CMD_ERASEUSERPROGRAM:     DINT := 6018;    (* Erase User Program *)
    MIO_CMD_SETUID:               DINT := 6019;    (* Set the unique ID of the module *)
    MIO_CMD_GETNBFREELOGITEMS:    DINT := 6020;    (* Return the number of free logbook items *)
    MIO_CMD_GETERRORCODE:         DINT := 6021;    (* Get the actual error code *)
    MIO_CMD_PERFORMEXTMEMTST:     DINT := 6022;    (* Test the external memories *)
    MIO_CMD_SAFETYGETVERSION_B:   DINT := 6023;    (* Get the version of the second processor *)
    MIO_CMD_SAFETYMEASWDGTIME:    DINT := 6024;    (* Measure the watchdog TIME OF the two processors *)

    (* Possible commands for the IO module TI214 *)
    MIO_CMD_SETAVERAGING:         DINT := 7001;    (* Set number of measure values for averging *)
    MIO_CMD_GETAVERAGING:         DINT := 7002;    (* Get number of measure values for averging *)

    (* Possible commands for the IO module FX2XX *)
	MIO_CMD_FMBASE:         DINT := 7200;
	MIO_CMD_GETSUPPLY:      DINT := 7201;   (* Transceiver Supply *)
	MIO_CMD_GETTXBIAS:      DINT := 7202;   (* TX Bias *)
	MIO_CMD_GETTXPOWER:     DINT := 7203;   (* TX Output Power *)
	MIO_CMD_GETRXPOWER:     DINT := 7204;   (* RX Output Power *)
	MIO_CMD_GETSCALEVALUES: DINT := 7205;   (* Get scale Values for Fibre Diagnosis *)
	MIO_CMD_SETSCALEVALUES: DINT := 7206;   (* Set scale Values for Fibre Diagnosis *)
	MIO_CMD_GETTHRESHOLD:   DINT := 7207;   (* Get FO thresholds *)
	MIO_CMD_GETCABLETYPE:   DINT := 7208;   (* get configured (jumper) cable type *)
	MIO_CMD_REINITFM:       DINT := 7220;   (* For internal use only: Reinit Fastbus Master *)
	MIO_CMD_RESETFM:        DINT := 7221;   (* For internal use only: Resets Fastbus Master *)

	(* Commands for the IO module FCS214 *)
	MIO_CMD_DIAG_GET_LNK:		   DINT := 7301; (* Get the link status for a port *)
	MIO_CMD_DIAG_GET_DUPLEX:	   DINT := 7302; (* Get the duplexity for a port *)
	MIO_CMD_DIAG_GET_SPEED: 	   DINT := 7303; (* Get the speed for a port *)
	MIO_CMD_DIAG_BAD_TRAFFIC_IN:   DINT := 7304; (* Get the sum of bytes of bad Frames for a port *)
	MIO_CMD_DIAG_TRAFFIC_IN:       DINT := 7305; (* Get the sum of bytes of good incoming Frames for a port *)
	MIO_CMD_DIAG_TRAFFIC_OUT:      DINT := 7306; (* Get the sum of bytes of outgoing Frames for a port *)
	MIO_CMD_SETTRIGERVALUES:       DINT := 7307; (* write the interrupt level value *)
	MIO_CMD_SETRESETCAPABILITY:	   DINT := 7308; (* Set modules reset capability *)
	MIO_CMD_GETRESETCAPABILITY:    DINT := 7309; (* Get modules reset capability *)
	MIO_CMD_GETMIRRORCFG: 		   DINT := 7310; (* Get Mirror Configuration *)
	MIO_CMD_SETMIRRORCFG: 		   DINT := 7311; (* Set Mirror Configuration *)

	(* Possible commands for the IO module ECS200 *)
	MIO_CMD_ECSBASE:        		DINT  := 7500;
	MIO_CMD_GETSLAVEINFO:   		DWORD := 16#00001d4d;

	(* Possible commands for the IO modules GIO2XX and AIO2XX *)
	MIO_CMD_GIOSETDOPULSE:          DWORD := 16#00001e79;   (* Set the digital output pulse times *)
	MIO_CMD_GIOGETDOPULSE:          DWORD := 16#00001e7a;   (* Read the digital output pulse times *)
	MIO_CMD_GIOSETAIFILTER:         DWORD := 16#00001e7b;   (* Set the analog input filter frequency *)
	MIO_CMD_GIOGETAIFILTER:         DWORD := 16#00001e7c;   (* Read the analog input filter frequency *)
	MIO_CMD_GIOSETSPIKEFILTER:      DWORD := 16#00001e7d;   (* Set the spike filter value *)
	MIO_CMD_GIOGETSPIKEFILTER:      DWORD := 16#00001e7e;   (* Read the spike filter value *)
	MIO_CMD_GIOSETLIMITS:           DWORD := 16#00001e7f;   (* Set analog input limits *)
	MIO_CMD_GIOGETLIMITS:           DWORD := 16#00001e80;   (* Read analog input limits *)
	MIO_CMD_GIOGETCHIPTEMP:         DWORD := 16#00001E81;   (* Read chip temperature *)
	MIO_CMD_GIOSETCOLDJUNCTEMP:     DWORD := 16#00001E82;   (* Set cold junction temperature *)
	MIO_CMD_GIOGETCOLDJUNCTEMP:     DWORD := 16#00001e83;   (* Read last set cold junction temperature *)
	MIO_CMD_GIOSETPWMRUNMODE:       DWORD := 16#00001e84;   (* Set the PWM run mode *)
	MIO_CMD_GIOGETPWMRUNMODE:       DWORD := 16#00001e85;   (* Read the PWM run mode *)
	MIO_CMD_GIOSETFILTERHB:         DWORD := 16#00001E86;   (* Activate or deactivate halfband filter *)
	MIO_CMD_GIOGETFILTERHB:         DWORD := 16#00001E87;   (* Get halfband filter setting *)
	MIO_CMD_GIOSETFILTERITP:        DWORD := 16#00001e88;   (* Activate or deactivate filter interpolation *)
	MIO_CMD_GIOGETFILTERITP:        DWORD := 16#00001e89;   (* Get filter interpolation setting *)
	MIO_CMD_GIOSETGROUNDED:         DWORD := 16#00001E8A;   (* Activate or deactivate grounded measurement *)
	MIO_CMD_GIOGETGROUNDED:         DWORD := 16#00001E8B;   (* Get activated or deactivated grounded measurement *)
	MIO_CMD_GIOGETNBRFIFOENTRIES:   DWORD := 16#00001E8C;   (* Get number of FIFO entries in counter and frequency modulation mode *)
	MIO_CMD_GIOGETFIFOVALUES:       DWORD := 16#00001E8D;   (* Get stored counter values from the FIFO in counter mode *)
	MIO_CMD_GIOGETFIFOOVERFLOW:     DWORD := 16#00001E8E;   (* Get number of overflows in the counter FIFO in counter mode *)
	MIO_CMD_GIOFIFOFLUSH:           DWORD := 16#00001E8F;   (* Flushes the FIFO in counter and frequency modulation mode *)
	MIO_CMD_GIOFIFOREFVALUE:        DWORD := 16#00001E90;   (* Get the reference value when FIFO started in counter mode *)
	MIO_CMD_GIOSTARTSTOPFIFO:       DWORD := 16#00001E91;   (* Starts/stops the FIFO in frequency modulation mode *)
	MIO_CMD_GIOSETPULSECOUNT:       DWORD := 16#00001E92;   (* Sets the pulse counter in frequency modulation mode *)
	MIO_CMD_GIOGETPULSECOUNT:       DWORD := 16#00001E93;   (* Gets the pulse counter in frequency modulation mode *)
	MIO_CMD_GIOSETPERIOD:           DWORD := 16#00001E94;   (* Sets the period in ns in pulse modulation mode *)
	MIO_CMD_GIOGETPERIOD:           DWORD := 16#00001E95;   (* Gets the period in ns in pulse modulation mode *)
	MIO_CMD_GIOADDFIFOENTRY:        DWORD := 16#00001E96;   (* Add a single FIFO entry in FIFO mode *)
	MIO_CMD_GIOSETPTCURRENT:        DWORD := 16#00001E97;   (* Set PT current *)
	MIO_CMD_GIOGETPTCURRENT:        DWORD := 16#00001E98;   (* Get PT current *)
	MIO_CMD_GIOSTARTSTOPFIFOEXT:    DWORD := 16#00001E99;   (* Starts/stops various channels using the FIFO for measurements *)

	(* AI208/SI specific filter constants *)
	MIO_AI_FILTER_2553:      DWORD := 16#0000;     (* 2553.13 *)
	MIO_AI_FILTER_1277:      DWORD := 16#0001;     (* 1277.06 *)
	MIO_AI_FILTER_639:       DWORD := 16#0002;     (* 638.52 *)
	MIO_AI_FILTER_319:       DWORD := 16#0003;     (* 319.26 *)
	MIO_AI_FILTER_160:       DWORD := 16#0004;     (* 159.63 *)
	MIO_AI_FILTER_80:        DWORD := 16#0005;     (* 79.81 *)
	MIO_AI_FILTER_40:        DWORD := 16#0006;     (* 39.91 *)
	MIO_AI_FILTER_20:        DWORD := 16#0007;     (* 19.95 *)
	MIO_AI_FILTER_10:        DWORD := 16#0008;     (* 9.98 *)
	MIO_AI_FILTER_5:         DWORD := 16#0009;     (* 4.99 *)
	MIO_AI_FILTER_2:         DWORD := 16#000A;     (* 2.49 *)

	(* GIO2xx specific filter constants *)
    (* Analog input filter frequencies *)
	MIO_GIO_AIFILTER_4kHz:      DWORD := 16#0;  (* Filter Frequency 4kHz *)
	MIO_GIO_AIFILTER_2kHz:      DWORD := 16#1;  (* Filter Frequency 2kHz *)
	MIO_GIO_AIFILTER_1kHz:      DWORD := 16#2;  (* Filter Frequency 1kHz *)
	MIO_GIO_AIFILTER_500Hz:     DWORD := 16#3;  (* Filter Frequency 500Hz *)
	MIO_GIO_AIFILTER_250Hz:     DWORD := 16#4;  (* Filter Frequency 250Hz *)
	MIO_GIO_AIFILTER_125Hz:     DWORD := 16#5;  (* Filter Frequency 125Hz *)
	MIO_GIO_AIFILTER_62_5Hz:    DWORD := 16#6;  (* Filter Frequency 62.5Hz *)
	MIO_GIO_AIFILTER_31_2Hz:    DWORD := 16#7;  (* Filter Frequency 31.2Hz *)
	MIO_GIO_AIFILTER_15_6Hz:    DWORD := 16#8;  (* Filter Frequency 15.6Hz *)
	MIO_GIO_AIFILTER_7_8Hz:     DWORD := 16#9;  (* Filter Frequency 7.8Hz *)
	MIO_GIO_AIFILTER_3_9Hz:     DWORD := 16#a;  (* Filter Frequency 3.9Hz *)
	MIO_GIO_AIFILTER_1_9Hz:     DWORD := 16#b;  (* Filter Frequency 1.9Hz *)
	MIO_GIO_AIFILTER_0_97Hz:    DWORD := 16#c;  (* Filter Frequency 0.97Hz *)
	MIO_GIO_AIFILTER_0_50Hz:    DWORD := 16#d;  (* Filter Frequency 0.50Hz *)

    (* Possible spike filter values *)
	MIO_GIO_SPIKEFILTER_OFF:    DWORD := 16#0000; (* Spike filter OFF *)
	MIO_GIO_SPIKEFILTER_16us:   DWORD := 16#1;    (* Spike filter 16us *)
	MIO_GIO_SPIKEFILTER_32us:   DWORD := 16#2;    (* Spike filter 32us *)
	MIO_GIO_SPIKEFILTER_64us:   DWORD := 16#3;    (* Spike filter 64us *)
	MIO_GIO_SPIKEFILTER_128us:  DWORD := 16#4;    (* Spike filter 128us *)
	MIO_GIO_SPIKEFILTER_256us:  DWORD := 16#5;    (* Spike filter 256us *)
	MIO_GIO_SPIKEFILTER_512us:  DWORD := 16#6;    (* Spike filter 512us *)
	MIO_GIO_SPIKEFILTER_1ms:    DWORD := 16#0007; (* Spike filter 1ms *)
	MIO_GIO_SPIKEFILTER_2ms:    DWORD := 16#0008; (* Spike filter 2ms *)
	MIO_GIO_SPIKEFILTER_4ms:    DWORD := 16#0009; (* Spike filter 4ms *)
	MIO_GIO_SPIKEFILTER_8ms:    DWORD := 16#000A; (* Spike filter 8ms *)
	MIO_GIO_SPIKEFILTER_16ms:   DWORD := 16#000B; (* Spike filter 16ms *)
	MIO_GIO_SPIKEFILTER_32ms:   DWORD := 16#000C; (* Spike filter 32ms *)
	MIO_GIO_SPIKEFILTER_65ms:   DWORD := 16#000D; (* Spike filter 65ms *)
	MIO_GIO_SPIKEFILTER_131ms:  DWORD := 16#000E; (* Spike filter 131ms *)
	MIO_GIO_SPIKEFILTER_262ms:  DWORD := 16#000F; (* Spike filter 262ms *)

	(* Error codes  *)
	MIO_ER_OK:                 DINT :=   0;    (* No error *)
	MIO_ER_FAIL:               DINT :=  -1;   (* General error *)
	MIO_ER_BADCHAN:            DINT :=  -2;   (* Channel NOT valid *)
	MIO_ER_BADMODE:            DINT :=  -3;   (* Mode OR TYPE NOT valid *)
	MIO_ER_BUSY:               DINT :=  -4;   (* Device is busy *)
	MIO_ER_BADTEST:            DINT :=  -5;   (* HwTest failed *)
	MIO_ER_BADCMD:             DINT :=  -6;   (* Command NOT supported *)
	MIO_ER_BADIDREG:           DINT :=  -7;   (* ID Register NOT valid *)
	MIO_ER_BADCONF:            DINT :=  -8;   (* Bad configuration *)
	MIO_ER_BADPARM:            DINT :=  -9;   (* Bad parameter *)
	MIO_ER_TIMEOUT:            DINT := -10;  (* Timeout *)
	MIO_ER_BADFUNC:            DINT := -11;  (* FUNCTION NOT supported *)
	MIO_ER_BADWRITE:           DINT := -12;  (* Error in write *)
	MIO_ER_NOWRITE:            DINT := -13;  (* Write on input channel *)
	MIO_ER_BADCALIB:           DINT := -14;  (* Bad calibration data *)
	MIO_ER_BADPLAUS:           DINT := -15;  (* Plausibility test failed *)
	MIO_ER_BADREAD:            DINT := -16;  (* Error in read *)
	MIO_ER_REBOOT:             DINT := -17;  (* Reboot is required *)
	MIO_ER_DISABLED:           DINT := -18;  (* Channel is disabled *)
	MIO_ER_WRONGSTATE:         DINT := -19;  (* Invalid state for this FUNCTION *)
	MIO_ER_BADCARD:            DINT := -20;  (* Card NOT valid *)
	MIO_ER_BUSFAIL:            DINT := -21;  (* Bus error *)
	MIO_ER_NODATA:             DINT := -22;  (* No data available *)
	MIO_ER_OUTOFMEM:           DINT := -23;  (* No memory available *)
	MIO_ER_NOFPTASK:           DINT := -24;  (* No floating point operations allowed *)
	MIO_ER_MODNOTINIT:         DINT := -25;  (* Module is NOT initialized *)
	MIO_ER_BADHANDLE:          DINT := -26;  (* Bad handle *)
	MIO_ER_LSTINFPGAFULL:      DINT := -27;  (* The list in the FPGA is full *)
	MIO_ER_WRONGITEMSIZE:      DINT := -28;  (* The DMA item has a wrong size *)
	MIO_ER_SEMCREATE:          DINT := -29;  (* Error creating a semaphore *)
	MIO_ER_SEMTAKE:            DINT := -30;  (* Error / Timeout taking a semaphore *)
	MIO_ER_WRONGMEMAREA:       DINT := -31;  (* Wrong memory area passed TO FUNCTION *)
	MIO_ER_BADALIGNMENT:       DINT := -32;  (* Bad alignment *)
	MIO_ER_UPDATELISTFULL:     DINT := -33;  (* Update list is full *)
	MIO_ER_WRONGPRIO:          DINT := -34;  (* Wrong priority *)
	MIO_ER_CHANNOTMAPPED:      DINT := -35;  (* Channel is NOT mapped *)
	MIO_ER_NOPIDRVID:          DINT := -36;  (* A process image module handle was expected but NOT given *)
	MIO_ER_HANDLEINUSE:        DINT := -37;  (* The actual handle is already in use *)
	MIO_ER_BIOSFAIL:           DINT := -38;  (* BIOS on module NOT running *)
	MIO_ER_DOWNGRADE:          DINT := -39;  (* Software downgrade *)
	MIO_ER_BADFIRMWARE:        DINT := -40;  (* Firmware doesn't fit on module *)
	MIO_ER_BADTYPE:            DINT := -41;  (* Module TYPE AND software TYPE are NOT compatible *)
	MIO_ER_NOAPP:              DINT := -42;  (* Application NOT found/registered *)
	MIO_ER_NOSCALEINF:         DINT := -43;  (* No scale information given for that channel *)
	MIO_ER_WRONGFUNCTYPE:      DINT := -44;  (* Wrong FUNCTION TYPE *)
	MIO_ER_NOTPRESENT:         DINT := -45;  (* Channel does NOT exist *)
	MIO_ER_OVERFLOW:           DINT := -46;  (* Channel value overflow *)
	MIO_ER_POWER:              DINT := -47;  (* Power failure *)

	(* Possible values for MIO_PROGRESS_R.Status *)
	PROGRESS_UNKNOWN:   DWORD := 16#00;
	PROGRESS_WORK:      DWORD := 16#01;
	PROGRESS_DONE:      DWORD := 16#02;
	PROGRESS_FAILED:    DWORD := 16#04;

END_VAR

(* Data type *)
TYPE GIO_DOPULSETIME :
STRUCT
    Period:     DINT;           (* Period length in us *)
    PulseWidth: DINT;           (* Pulse width (0% .. 100% -> 0 .. 65535) *)
    StartPulse: DINT;           (* Start pulse time in us *)
END_STRUCT
END_TYPE

(* Data type *)
TYPE LOGIC_VERSION (* HW version *)
STRUCT
	TestVer: BYTE;            (* Testversion *)
	Revision: BYTE;           (* Revision number *)
 	Design: UINT;             (* Hardware design number *)
	Ver32: UDINT;             (* 32-Bit Version *)
END_STRUCT
END_TYPE

(* Data type *)
TYPE MIO_ACRERR	(* used with Mio_DoCmd4() and Mio_CMD_GetVal/SetVal for ACR222 *)
STRUCT							(* structure for error-information of ACR222-Card *)
	Index:			WORD;		(* affected Object-Index *)
	SubIndex:		WORD;		(* affected Object-SubIndex *)
	AddCode:		WORD;		(* meaning of AddCode, ErrorCode *)
	ErrorCode:	BYTE;			(* and ErrorClass see "CiA DS 301", *)
	ErrorClass:	BYTE;			(* chapter "The Service Data Object" *)
END_STRUCT
END_TYPE

(* Data type *)
(* part of return-structure of Mio_GetExtCardInf *)
TYPE MIO_CLOCK
STRUCT
    Second: DINT;		(* range 0 - 59 *)
    Minute: DINT;		(* range 0 - 59 *)
    Hour: DINT;			(* range 0 - 23 *)
    Day: DINT;			(* range 1 - 31 *)
    Month: DINT;		(* range 0 - 11 *)
    Year: DINT;			(* years since 1900 *)
    WeekDay: DINT;	(* range 0 = Sunday ... 6 = Saturday *)
    YearDay: DINT;		(* range 0 - 365 *)
    DSTFlag: DINT;		(* DayLightSaving-Time Flag *)
END_STRUCT
END_TYPE

(* Data type *)
(* Return structure of Mio_GetInterruptInfo *)
TYPE MIO_INTINFO
STRUCT
	CardNb:  DINT;			(* The Card-Number of the Card that caused the interrupt(Only valid		*)
							(* for a Event or Error Interrupt)										*)
	ChanNb:  DINT;			(* The Channel-Number of the channel that caused the interrupt(Only		*)
							(* valid for a Event or Error Interrupt)								*)
							(* 0   = Interrupt caused by module										*)
							(* 1-n = Interrupt caused by given channel								*)
	Mask:	DWORD;			(* Gives the bit mask of the Event or Error Interrupt					*)
							(* For an Error Interrupt, use the Mio_ERR_* constants to mask out values	*)
							(* For an Event Interrupt, use the Mio_EVT_* constants to mask out values	*)
	Spare0: DWORD;			(* reserved *)
	Spare1: DWORD;			(* reserved *)
	Spare2: DWORD;			(* reserved *)
	Spare3: DWORD;			(* reserved *)
END_STRUCT
END_TYPE

(* Data type *)
TYPE MIO_MINMAX (* Structure for Mio_SetMinMaxXXX and Mio_GetMinMaxEvent on AI204 *)
STRUCT
	MinVal: DINT;		(* Minumum value *)
	MaxVal: DINT;		(* Maximum value *)
END_STRUCT
END_TYPE

(* Data type *)
TYPE MIO_RETCARDINF		(* return-structure of Mio_GetCardInf *)
STRUCT
	RetCode: DINT;			(*  Success (0) - or Error-Code (<0) *)
	CardNb: DINT;			(* Card-Number *)
	CardType: DINT;			(* Card-Type *)
	CardVariant: DINT;		(* Card-Variant *)
	CardCategory: DWORD;	(* Card-Category *)
	CardFlags: DWORD;		(* Properies of Card *)
	MaxChan: DINT;			(* number of Channels *)
END_STRUCT
END_TYPE

(* Data type *)
TYPE MIO_RETCHANINF		(* return-structure of Mio_GetChanInf *)
STRUCT
	RetCode: DINT;			(*  Success (0) - or Error-Code (<0) *)
	ChanCategory: DWORD;	(* Channel-Category *)
	ChanFlags: DWORD;		(* Properies of Channel *)
END_STRUCT
END_TYPE

(* Data type *)
TYPE MIO_RETCHANRANGEINF		(* return-structure of Mio_GetChanRangeInf *)
STRUCT
    RetCode: DINT;			           (* Success (0) - or Error-Code (<0) *)
    DispMode : UDINT;                  (* Display Mode: UFB_DISP_MODE (default: UFB_DISP_MODE_RAW_DEZ) *)
    Range : UDINT;                     (* Range code OF channel (MIO_R_NONE, MIO_R16_20MA, ...) *)
    Scale : LREAL;                     (* Scaling factor (default: 1.0) *)
    Offset : LREAL;                    (* Offset (default: 0.0) *)
    MeasuringMin : REAL;               (* Measuring range minimum (e.g. AI208 = -25mA) *)
    MeasuringMax : REAL;               (* Measuring range maximum (e.g. AI208 = +25mA) *)
    ConfigMin : REAL;                  (* Scaled minimum value (e.g. AI208 = +4mA) *)
    ConfigMax : REAL;                  (* Scaled maximum value (e.g. AI208 = +20mA) *)
    RawMinLow :  UDINT;                (* Raw minimum value (e.g. AI208 = 0) low UDINT *)
    RawMinHigh : UDINT;                (* Raw minimum value (e.g. AI208 = 0) high UDINT *)
    RawMaxLow :  UDINT;                (* Raw maximum value (e.g. AI208 = 65535) low UDINT *)
    RawMaxHigh : UDINT;                (* Raw maximum value (e.g. AI208 = 65535) high UDINT *)
    len : UDINT;                       (* Size OF raw value in bytes (normally 4) *)
    Format : UDINT;                    (* SVI format OF value (normally SVI_F_SINT32) *)
    BaseSiUnit : UDINT;                (* SI-Unit: UFB_SIUNIT (default: UFB_SIUNIT_NONE) *)
    BaseUnitStr : STRING(11);          (* Physical unit base optional text (e.g. "V", "RPM", "A" ATTENTION: NOT "mA") *)
    BasePrefixFactor : DINT;           (* Exponent TO the base 10 OF the unit (e.g. -3 FOR mA) *)
    ExtChFlags : UINT;                 (* Extended channel flags (MIO_EXTFLG_* ) *)
    Spare : ARRAY[1..31] OF UINT;      (* Spare FOR future extension *)
END_STRUCT
END_TYPE

(* Data type *)
TYPE MIO_RETEXTCARDINF	(* return-structure of Mio_GetExtCardInf *)
STRUCT
	RetCode: DINT;			(*  Success (0) - or Error-Code (<0) *)
	CardNb: DINT;			(* Card-Number *)
	StationNb: DINT;		(* Station-Number *)
	SlotNb: DINT;			(* Slot-Number *)
	PreSlots: DINT;			(* precessing- *)
	PostSlots: DINT;		(* + following-also-used-slots *)
	Mode: DINT;				(* Mode of Card-Driver *)
	State: DINT;			(* State of Card-Driver *)
	CardType: DINT;			(* Card-Type *)
	CardVariant: DINT;		(* Card-Variant *)
	CardCategory: DWORD;	(* Card-Category *)
	CardFlags: DWORD;		(* Properies of Card *)
	MaxChan: DINT;			(* number of Channels *)
	Version: DINT;			(* Card-Version *)
	DrvVersion: DINT;		(* necc. Driver-Version *)
	Attribute: DWORD;		(* defined/set  Attributes *)
	ProdTime: MIO_CLOCK;	(* Date + Time of production *)
	ProdNb: STRING(11);		(* Serial-No.-String *)
	Name: STRING(23);		(* Name of Card *)
	Info: STRING(199);		(* Block of Info-Text *)
	DrvName: STRING(15);	(* Name of Driver-*.M-File *)
	Power: DINT;				(* Power consumption in [mW] *)
	Reserved: STRING(35);	(* reserved for future use *)
END_STRUCT
END_TYPE

(* Data type *)
TYPE MIO_RETEXTCARDINF2	(* return-structure of Mio_GetExtCardInf *)
STRUCT
	RetCode: DINT;			(*  Success (0) - or Error-Code (<0) *)
	CardNb: DINT;			(* Card-Number *)
	StationNb: DINT;		(* Station-Number *)
	SlotNb: DINT;			(* Slot-Number *)
	PreSlots: DINT;			(* precessing- *)
	PostSlots: DINT;		(* + following-also-used-slots *)
	Mode: DINT;				(* Mode of Card-Driver *)
	State: DINT;			(* State of Card-Driver *)
	CardType: DINT;			(* Card-Type *)
	CardVariant: DINT;		(* Card-Variant *)
	CardCategory: DWORD;	(* Card-Category *)
	CardFlags: DWORD;		(* Properies of Card *)
	MaxChan: DINT;			(* number of Channels *)
	Version: DINT;			(* Card-Version *)
	DrvVersion: DINT;		(* necc. Driver-Version *)
	Attribute: DWORD;		(* defined/set  Attributes *)
	ProdTime: MIO_CLOCK;	(* Date + Time of production *)
	ProdNb: STRING(11);		(* Serial-No.-String *)
	Name: STRING(23);		(* Name of Card *)
	Info: STRING(199);		(* Block of Info-Text *)
	DrvName: STRING(15);	(* Name of Driver-*.M-File *)
	Power: DINT;	    	(* Power consumption in [mW] *)
 	Current_5V: DINT;       (* 5V Current sink/source in mA *)
    Current_P15V: DINT;     (* +15V Current sink/source in mA *)
    Current_M15V: DINT;     (* -15V Current sink/source in mA *)
    ModVerType: DINT;       (* Version Type code MIO_VER_ *)
    RedundantRead: BOOL;    (* Redundant read of data if TRUE *)
    WriteVerify: BOOL;      (* Write verify of data if TRUE *)
    BusCheck: BOOL;         (* BUSCHECK supported if TRUE *)
    AliveCheck: BOOL;       (* ALIVECHECK supported if TRUE *)
    AssemblyCode: WORD;     (* Function code lower part *)
    HwVariant: BYTE;        (* Hardware variant *)
    Reserved1: BYTE;        (* Not used, 0 for now *)
    Settings: DWORD;        (* Flags that may be en-/disabled *)
    ExStateInfo: DWORD;     (* Extended state information *)
    Versions: MIO_VERSION;  (* Versions OF this module (FW, Logic, ...) *)
    PackageVers: MIO_VERS;  (* Package version *)
    PartNumber: UDINT;      (* Part number (0 IF NOT available) *)
    FirmBackup: BOOL;       (* Firmware can be recovered *)
    Spare1: ARRAY [1..3] OF BYTE;   (* Align it TO 32 bit *)
 	Spare: ARRAY [1..29] OF UDINT;  (* NOT used, 0 FOR now *)

END_STRUCT
END_TYPE

(* Data type *)
TYPE MIO_RETFOUND	(* return-structure of Mio_GetNextError *)
STRUCT
	RetCode: DINT;		(*  Success (0 or 1) - or Error-Code (<0) *)
	Card: DINT;			(*  Card with Error (-1 for None)  (valid in case of Success) *)
	Chan: DINT;			(*  Chan with Error (-1 for None) (valid in case of Success) *)
	State: DWORD;		(*  Error-State (valid in case of Success) *)
END_STRUCT
END_TYPE

(* Data type *)
TYPE MIO_RETSCALEINF :
STRUCT
	RetCode		: DINT;		(* Success- or Error-Code *)
	ScaleInf	: DWORD;	(* Return-Pointer to Scale information of the channel *)
END_STRUCT
END_TYPE

(* Data type *)
TYPE MIO_RETSTATE	(* return-structure used by Mio_GetError, -Select, -Chan- and -CardMode *)
STRUCT
	RetCode: DINT;		(* Success- or Error-Code *)
	State: DWORD;		(* depending on returning function: Error-State, Select-Info or Chan/Card-Mode *)
END_STRUCT
END_TYPE

(* Data type *)
TYPE MIO_RETVALUE	(* return-structure of Mio_GetValue *)
STRUCT
	RetCode: DINT;		(* Success- or Error-Code *)
	Value: DINT;			(* IO-Value (valid in case of Success) *)
END_STRUCT
END_TYPE

(* Data type *)
TYPE MIO_RETVALUE_LREAL :
STRUCT
	RetCode: DINT;		(* Success- or Error-Code *)
	Value: LREAL;			(* IO-Value (valid in case of success) *)
END_STRUCT
END_TYPE

(* Data type *)
TYPE MIO_VERS (* Version information *)
STRUCT
	Major: BYTE;     (* Major Version        V.xx.xx *)
	Minor: BYTE;     (* Minor Version        x.VV.xx *)
	SubMin: BYTE;    (* Sub-Minor Version    x.xx.VV *)
	VerType: BYTE;   (* M_VER_ALPHA, M_VER_BETA or M_VER_RELEASE *)
	Ver32: UDINT;    (* 32-Bit Version *)
END_STRUCT
END_TYPE

(* Data type *)
TYPE MIO_VERSION (* Structure for I/O module versions *)
STRUCT
 	Driver: SYS_VERSION;            (* Version OF MIO-Driver *)
    Fware: SYS_VERSION;             (* Version of Firmware *)
    Bios: SYS_VERSION;              (* Version of BIOS *)
    Logic: LOGIC_VERSION;           (* Logic Version (since MBase 3.90) *)
	Spare: ARRAY [1..12] OF BYTE;   (* Filled with zero FOR now *)
END_STRUCT
END_TYPE

(* Data type *)
TYPE SYS_VERSION (* Version code, do not change values or size of this structure *)
STRUCT
	Code: ARRAY [1..3] OF UDINT;   (* Version code OF object *)
    SysType: UDINT;                (* Version type of object *)
END_STRUCT
END_TYPE

(* POU Mio_AttachError, IL *)
(******************************************************************************
Description: Attaches attention to an error of an IO-card / channel
Input:
  - CardId: ID of the card
  - Chan: Channel number
  - Error:  Bitcoded error-cases to pay attention to 
Return: 
  - DINT => Success- or error-code
******************************************************************************)
FUNCTION Mio_AttachError : DINT
VAR_INPUT
	CardId: DINT;
	Chan: DINT;
	Error: DWORD;		(* Bitcoded error-cases to pay attention to *)
END_VAR
LD 0
END_FUNCTION

(* POU Mio_BadCustomerID, ST *)
FUNCTION Mio_BadCustomerID : DINT
VAR_INPUT
	CardId: DINT;
	LogError: BOOL;
END_VAR
VAR
END_VAR
;
END_FUNCTION

(* POU Mio_CalcRawValueDINT2DINT, ST *)
(******************************************************************************
Description: Calculate the raw value of a channel from the given 
			 scaled value with type DINT to the result type DINT.
Input:
  - ScaleInf:  Handle to Scale information of the channel.
  - Value:     Scaled value to perform inverse scaling.
Return: 
  - MIO_RETVALUE.RetCode: DINT => Success- or error-code
  - MIO_RETVALUE.Value:	  DINT => Calculated raw value (valid in case of success)
******************************************************************************)
FUNCTION Mio_CalcRawValueDINT2DINT : MIO_RETVALUE
VAR_INPUT
	ScaleInf	: DWORD;		(* Pointer to Scale information of the channel *)
	Value	: DINT;		        (* input: scaled value  *)
END_VAR
VAR
END_VAR
;
END_FUNCTION

(* POU Mio_CalcRawValueLREAL2DINT, ST *)
(******************************************************************************
Description: Calculate the raw value of a channel from the given 
			 scaled value with type LREAL to the result type DINT.

Input:
  - ScaleInf:  Handle to Scale information of the channel.
  - Value:     Scaled value to perform inverse scaling.
Return: 
  - MIO_RETVALUE.RetCode: DINT => Success- or error-code
  - MIO_RETVALUE.Value:	  DINT => Calculated raw value (valid in case of success)
******************************************************************************)
FUNCTION Mio_CalcRawValueLREAL2DINT : MIO_RETVALUE
VAR_INPUT
	ScaleInf 	: DWORD;	(* Pointer to Scale information of the channel *)
	Value	: LREAL;		(* Input: scaled value  *)
END_VAR
VAR
END_VAR
;
END_FUNCTION

(* POU Mio_CalcRawValueLREAL2LREAL, ST *)
(******************************************************************************
Description: Calculate the raw value of a channel from the given 
			 scaled value with type LREAL to the result type LREAL.

Input:
  - ScaleInf:  Handle to Scale information of the channel.
  - Value:     Scaled value to perform inverse scaling.
Return: 
  - MIO_RETVALUE_LREAL.RetCode: DINT => Success- or error-code
  - MIO_RETVALUE_LREAL.Value:	LREAL => Calculated raw value 
                                (valid in case of success)
******************************************************************************)
FUNCTION Mio_CalcRawValueLREAL2LREAL : MIO_RETVALUE_LREAL
VAR_INPUT
	ScaleInf 	: DWORD;		(* Pointer to Scale information of the channel *)
	Value	: LREAL;		    (* input: scaled value  *)
END_VAR
VAR
END_VAR
;
END_FUNCTION

(* POU Mio_CalcScaledValueDINT2DINT, ST *)
(******************************************************************************
Description: Calculate the scaled value of a channel from the given 
             raw value with type DINT to the result type DINT.
Input:
  - ScaleInf:  Handle to Scale information of the channel
  - Value:     Original value to perform  scaling
Return: 
  - MIO_RETVALUE.RetCode: DINT => Success- or error-code
  - MIO_RETVALUE.Value:	  DINT => Calculated scaled value (valid in case of success)
******************************************************************************)
FUNCTION Mio_CalcScaledValueDINT2DINT : MIO_RETVALUE
VAR_INPUT
	ScaleInf 	: DWORD;		(* Pointer to Scale information of the channel *)
	OrgVal	: DINT;			(* input: original value *)
END_VAR
VAR
END_VAR
;
END_FUNCTION

(* POU Mio_CalcScaledValueDINT2LREAL, ST *)
(******************************************************************************
Description: Calculate the scaled value of a channel from the given
             raw value with type DINT to the result type LREAL.
Input:
  - ScaleInf:  Handle to Scale information of the channel
  - Value:     Original value to perform  scaling
Return: 
Return: 
  - MIO_RETVALUE_LREAL.RetCode: DINT => Success- or error-code
  - MIO_RETVALUE_LREAL.Value:	LREAL => Calculated scaled value 
                                (valid in case of success)
******************************************************************************)
FUNCTION Mio_CalcScaledValueDINT2LREAL : MIO_RETVALUE_LREAL
VAR_INPUT
	ScaleInf 	: DWORD;	(* Pointer to Scale information of the channel *)
	OrgVal	: DINT;			(*input: original value *)
END_VAR
VAR
END_VAR
;
END_FUNCTION

(* POU Mio_CalcScaledValueLREAL2LREAL, ST *)
(******************************************************************************
Description: Calculate the scaled value of a channel from the given
             raw value with type LREAL to the result type LREAL.
Input:
  - ScaleInf:  Handle to Scale information of the channel
  - Value:     Original value to perform  scaling
Return: 
  - MIO_RETVALUE_LREAL.RetCode: DINT => Success- or error-code
  - MIO_RETVALUE_LREAL.Value:	LREAL => Calculated scaled value 
                                (valid in case of success)
******************************************************************************)
FUNCTION Mio_CalcScaledValueLREAL2LREAL : MIO_RETVALUE_LREAL
VAR_INPUT
	ScaleInf 	: DWORD;	(* Pointer to Scale information of the channel *)
	OrgVal	: LREAL;		(* Input: original value *)
END_VAR
VAR
END_VAR
;
END_FUNCTION

(* POU Mio_DetachError, IL *)
(******************************************************************************
Description: Detaches attention from an error of an IO-card / channel
Input:
  - CardId: The cards ID
  - Chan: Channel number
  - Error:  Bitcoded error-cases to detach attention from 
Return: 
  - DINT => Success- or error-code
******************************************************************************)
FUNCTION Mio_DetachError : DINT
VAR_INPUT
	CardId: DINT;
	Chan: DINT;
	Error: DWORD;		(* Bitcoded error-cases to detach attention from *)
END_VAR
LD 0
END_FUNCTION

(* POU Mio_DoCmd, IL *)
(******************************************************************************
Description: Executes a card specific function
Input:
  - CardId: ID of the card
  - Chan: Channel number
  - Cmd:  Card/driver command (specific)
  - ArgVal:  Additional parameter to command 
Return: 
  - DINT => Success- or error code
******************************************************************************)
FUNCTION Mio_DoCmd : DINT
VAR_INPUT
	CardId: DINT;
	Chan: DINT;
	Cmd: DWORD;			(* Card/driver command (specific) *)
	ArgVal: DWORD;		(* Additional parameter to command  *)
END_VAR
LD 0
END_FUNCTION

(* POU Mio_DoCmd4, IL *)
(******************************************************************************
Description: Executes a card specific function with 4 parameters
Input:
  - CardId: ID of the card
  - Chan: Channel number
  - Cmd:  Card/driver command (specific)
  - ArgVal1:  Additional parameter 1 to command 
  - ArgVal2:  Additional parameter 2 to command 
  - ArgVal3:  Additional parameter 3 to command 
  - ArgVal4:  Additional parameter 4 to command 
Return: 
  - DINT => Success- or error code
******************************************************************************)
FUNCTION Mio_DoCmd4 : DINT
VAR_INPUT
	CardId: DINT;
	Chan: DINT;
	Cmd: DWORD;		(* Card/driver command (specific) *)
	ArgVal1: DWORD;		(* Additional parameter 1 to command *)
	ArgVal2: DWORD;		(* Additional parameter 2 to command *)
	ArgVal3: DWORD;		(* Additional parameter 3 to command *)
	ArgVal4: DWORD;		(* Additional parameter 4 to command *)
END_VAR
	LD		0
END_FUNCTION

(* POU Mio_DoCmd8, IL *)
(******************************************************************************
Description: Executes a card specific function with 8 parameters
Input:
  - CardId: ID of the card
  - Chan: Channel number
  - Cmd:  Card/driver command (specific)
  - ArgVal1:  Additional parameter 1 to command 
  - ArgVal2:  Additional parameter 2 to command 
  - ArgVal3:  Additional parameter 3 to command 
  - ArgVal4:  Additional parameter 4 to command 
  - ArgVal5:  Additional parameter 5 to command 
  - ArgVal6:  Additional parameter 6 to command 
  - ArgVal7:  Additional parameter 7 to command 
  - ArgVal8:  Additional parameter 8 to command 
Return: 
  - DINT => Success- or error code
******************************************************************************)
FUNCTION Mio_DoCmd8 : DINT
VAR_INPUT
	CardId: DINT;
	Chan: DINT;
	Cmd: DWORD;		(* Card/driver command (specific) *)
	ArgVal1: DWORD;		(* Additional parameter 1 to command *)
	ArgVal2: DWORD;		(* Additional parameter 2 to command *)
	ArgVal3: DWORD;		(* Additional parameter 3 to command *)
	ArgVal4: DWORD;		(* Additional parameter 4 to command *)
	ArgVal5: DWORD;		(* Additional parameter 5 to command *)
	ArgVal6: DWORD;		(* Additional parameter 6 to command *)
	ArgVal7: DWORD;		(* Additional parameter 7 to command *)
	ArgVal8: DWORD;		(* Additional parameter 8 to command *)
END_VAR
LD 0
END_FUNCTION

(* POU Mio_DoCmd8_NB, ST *)
(******************************************************************************
Description: Executes a card specific function with 8 parameters (non-blocking)
Input:
  - Req:  		Request enable
  - CardId: 	ID of the card
  - Chan: 		Channel number
  - Cmd:  		Card/driver command (specific)
  - ArgVal1:  	Additional parameter 1 to command 
  - ArgVal2:  	Additional parameter 2 to command 
  - ArgVal3:  	Additional parameter 3 to command 
  - ArgVal4:  	Additional parameter 4 to command 
  - ArgVal5:  	Additional parameter 5 to command 
  - ArgVal6: 	Additional parameter 6 to command 
  - ArgVal7:  	Additional parameter 7 to command 
  - ArgVal8:  	Additional parameter 8 to command 
Output:
  - Done:  		TRUE => operation completed 
  - Error:  	TRUE in case of error 
  - ErrorId:  	0: OK/Done, 1: BUSY, Error-Code in case of error 

******************************************************************************)
FUNCTION_BLOCK Mio_DoCmd8_NB
VAR_INPUT
	Req : BOOL;
	CardId: DINT;
	Chan: DINT;
	Cmd: DWORD;
	ArgVal1: DWORD;
	ArgVal2: DWORD;
	ArgVal3: DWORD;
	ArgVal4: DWORD;
	ArgVal5: DWORD;
	ArgVal6: DWORD;
	ArgVal7: DWORD;
	ArgVal8: DWORD;
END_VAR
VAR_OUTPUT
	Done : BOOL;
	Error : BOOL;
	ErrorId : DINT;
END_VAR
VAR
	Pltd : DWORD;
END_VAR
;
END_FUNCTION_BLOCK

(* POU Mio_ExtractLibErr, ST *)
(******************************************************************************
Description: Most functions of the MIO-library, eg Mio_AttachError, return
             a 'packed' error-code which encodes two specific errors. 

             This function extracts the library-error of the encoded error. 
             The library-error is generated in the mio-library directly, 
             eg through checking the input-parameters. 

             The library-error can be compared against the Mio_ERC_xxx-constants. 
Input:
  - Error: error returned by the Mio_-function
Return: 
  - DINT, see description
******************************************************************************)

FUNCTION Mio_ExtractLibErr : DINT
VAR_INPUT
	Error: DINT;
END_VAR
VAR
END_VAR
;
END_FUNCTION

(* POU Mio_ExtractMioErr, ST *)
(******************************************************************************
Description: Most functions of the MIO-library, eg Mio_AttachError, return
             a 'packed' error-code which encodes two specific errors. 

             This function extracts the MIO-error (the error of the underlying mio-
             C-function) of the encoded error. 
Input:
  - Error: error returned by the Mio_-function
Return: 
  - DINT, see description
******************************************************************************)

FUNCTION Mio_ExtractMioErr : DINT
VAR_INPUT
	Error: DINT;
END_VAR
VAR
END_VAR
;
END_FUNCTION

(* POU Mio_GetBadSlaveReboot, ST *)
(******************************************************************************
Description: Returns the configuration for bad FAST Bus slave stations behaviour. 
Input:
  - Dummy: 
Return: 
  - TRUE: If the return value is TRUE, the controller will reboot as soon as a
    bad station is recognized.
  - FALSE: If the return value is FALSE, the complete chain of stations on
    that FM21x will be shut down and no reboot happens.
******************************************************************************)
FUNCTION Mio_GetBadSlaveReboot : BOOL
VAR_INPUT
	Dummy: DINT;
END_VAR
;
END_FUNCTION

(* POU Mio_GetBadStationList, ST *)
(******************************************************************************
Description: Indicates which stations are not available (shutdown). Bits 0-15
   correspond to stations 1-16, where a bit value of 1 indicates the
   station is "Bad" (not available).
Input:
  - Dummy: 
Return: 
  - 0: all Station are OK
  - 1-n: check bits 0-15 to see which stations are "Bad".
******************************************************************************)
FUNCTION Mio_GetBadStationList : DWORD
VAR_INPUT
	Dummy: DINT;
END_VAR
;
END_FUNCTION

(* POU Mio_GetBlk, IL *)
(******************************************************************************
Description: Reads a block value of a IO-channel
Input:
  - CardId: ID of the card
  - Chan: Channel number
  - pValue: Pointer to return buffer 
  - pLen: Amount of bytes to be read from buffer
Output:
  - pValue: Returned data
  - pLen: Returned block value length
Return: 
  - RetCode: DINT => Success- or error-code
******************************************************************************)
FUNCTION Mio_GetBlk : DINT
VAR_INPUT
	CardId: DINT;
	Chan: DINT;
	pValue: POINTER TO BYTE;
	pLen: POINTER TO UDINT;
END_VAR
LD 0
END_FUNCTION

(* POU Mio_GetCardInf, IL *)
(******************************************************************************
Description: Gets information of an IO-card
Input:
  - CardId: The ID of the card
Return: 
  - MIO_RETCARDINF.RetCode: DINT => Success- or error code
  - MIO_RETCARDINF.CardNb: DINT =>  Card number (valid in case of success)
  - MIO_RETCARDINF.CardType: DINT =>  Card type (valid in case of success)
  - MIO_RETCARDINF.CardVariant: DINT => Card variant (valid in case of success)
  - MIO_RETCARDINF.CardCategory: DWORD =>  Card category (valid in case of success)
  - MIO_RETCARDINF.CardFlags: DWORD =>  Properies of card (valid in case of success)
  - MIO_RETCARDINF.MaxChan: DINT =>  Number of channels (valid in case of success)
******************************************************************************)
FUNCTION Mio_GetCardInf : MIO_RETCARDINF
VAR_INPUT
	CardId: DINT;
END_VAR
LD 0
END_FUNCTION

